// TIA Portal project "ENSACADPORA_030924" (V18)

(* hardware
DEVICE "SIMATIC 1200 station_1"  S7-1200 Station
   slot 0: "S7-1200 rack"  S7-1200 Rack  Rack  V1.0
   slot 1: "Master"  CPU 1212C DC/DC/Rly  6ES7 212-1HE40-0XB0  V4.5
   slot 2: "DI 8x24VDC/DQ 8xRelay_1"  SM 1223 DI8/DQ8 x relay  6ES7 223-1PH32-0XB0  V2.0
   slot 101: "CM 1241 (RS422/485)_1"  6ES7 241-1CH32-0XB0  V2.2
*)

// ===== PLC "Master"  CPU 1212C DC/DC/Rly =====

VAR_GLOBAL   // PLC tag table "Default tag table"
   "Input_IniciarLLenado" AT %I0.0 : Bool;
   "Input_PararLLenado" AT %I0.1 : Bool;
   "Input_ParoEmergencia" AT %I0.2 : Bool;
   "Input_SensorInicioPistonComp" AT %I0.3 : Bool;
   "Input_SensorFinPistonComp" AT %I0.4 : Bool;
   "COM_ACTIVA" AT %M113.0 : Bool;
   "StepCom" AT %MB57 : Byte;
   "System_Byte" AT %MB58 : Byte;
   "FirstScan" AT %M50.0 : Bool;
   "DiagStatusUpdate" AT %M50.1 : Bool;
   "AlwaysTRUE" AT %M50.2 : Bool;
   "AlwaysFALSE" AT %M50.3 : Bool;
   "FrmHmi_EncenderMotorHelicoidal" AT %M60.0 : Bool;
   "FrmHmi_ApagarMotorHelicoidal" AT %M60.1 : Bool;
   "FrmHmi_ResetFallas" AT %M61.0 : Bool;
   "Refe_Frec_FromHmi_ToVdf" AT %MW0 : Int;
   "AuxIn_IniciarLLenado" AT %M56.0 : Bool;
   "AuxIn_PararLLenado" AT %M56.1 : Bool;
   "AuxIn_ParoEmergancia" AT %M56.2 : Bool;
   "AuxIn_SensorInicioComp" AT %M56.3 : Bool;
   "AuxIn_SensorFinalComp" AT %M56.4 : Bool;
   "FrmHmi_ModManual" AT %M63.0 : Bool;
   "FrmHmi_Automatico" AT %M63.1 : Bool;
   "FrmHmi_ActivarPistonCompuerta" AT %M60.2 : Bool;
   "FrmHmi_DesactivarPistonCompuerta" AT %M60.3 : Bool;
   "Aux_Modo_Manual" AT %M64.0 : Bool;
   "Aux_Modo_Auto" AT %M64.1 : Bool;
   "SetPoitKilos" AT %MD4 : Real;
   "FrmHmi_HacerZeroBas" AT %M60.7 : Bool;
   "PB POLARIDAD" AT %M65.0 : Bool;
   "BAS ESTABLE" AT %M65.1 : Bool;
   "BAS UNDERLOAD" AT %M65.2 : Bool;
   "BAS OVERLOAD" AT %M65.3 : Bool;
   "BAS TARA HECHA" AT %M65.4 : Bool;
   "BAS EN ZERO" AT %M65.5 : Bool;
   "PESO NETO BASCULA" AT %MD44 : Real;
   "FrmHmi_ActivarModBarrido" AT %M63.2 : Bool;
   "OUT_VDF_MOTOR" AT %Q0.0 : Bool;
   "OUT_VIBRADOR" AT %Q0.2 : Bool;
   "OUT_COMPUERTA_ABIERTA" AT %Q0.1 : Bool;
   "FrmHmi_EncenderVibradorEnsacadora" AT %M60.4 : Bool;
   "FrmHmi_ApagarVibradorEnsacadora" AT %M60.5 : Bool;
   "Aux_Modo_Barrido" AT %M64.2 : Bool;
   "FrmHmi_DesactivarModBarrido" AT %M63.3 : Bool;
   "AUX_OUT_MOTOR" AT %M66.0 : Bool;
   "AUX_OUT_VIBRADOR" AT %M66.1 : Bool;
   "AUX_OUT_COMPUERTA_ABIERTA" AT %M66.2 : Bool;
   "AUX_OUT_MOTOR_BARRIDO" AT %M66.3 : Bool;
   "AUX_OUT_VIBRADOR_BARRIDO" AT %M66.4 : Bool;
   "AUX_OUT_COMPUERTA_BARRIDO_ABIERTA" AT %M66.5 : Bool;
   "ESTATUS_OPERACION" AT %MW8 : Int;
   "FrmHmi_Barrido" AT %M63.4 : Bool;
   "AUX_PARO_EMERGENCIA" AT %M61.1 : Bool;
   "INCIAR CICLO" AT %M62.0 : Bool;
   "APAGAR CICLO" AT %M62.1 : Bool;
   "Aux_Reset_Ciclo" AT %M64.3 : Bool;
   "Aux Error COM bascula" AT %M64.4 : Bool;
   "Aux iniciar ciclo" AT %M64.5 : Bool;
   "STEP BASCULA" AT %MW10 : Int;
   "Aux Valvula compuerta de carga_abierta" AT %M64.6 : Bool;
   "Abriendo compuerta de carga" AT %M67.0 : Bool;
   "Aux Sensor Compuerta Carga Abierta" AT %M64.7 : Bool;
   "pasa o no pasa" AT %MW12 : Int;
   "PESO NETO" AT %MD40 : Real;
   "TARAR" AT %MD36 : Real;
   "aux zero manual" AT %M60.6 : Bool;
   "AUX_HACER_ZERO" AT %M65.6 : Bool;
   "ZERO RES" AT %M65.7 : Bool;
   "SETPOINT" AT %MW2 : Int;
   "ACTIVAR MOTOR" AT %M66.6 : Bool;
   "PUNTO DE CORTE" AT %MD32 : Real;
   "% Corte VFD Grueso" AT %MW14 : Int;
   "Frec Max Mot Fino" AT %MW16 : Int;
   "OUT FRECU PARA VDF FINO" AT %MW18 : Int;
   "DIFERENCIA" AT %MD28 : Real;
   "DIV" AT %MD20 : Real;
   "FILTRO" AT %MD24 : Real;
   "Aux falla arranque VDF" AT %M56.5 : Bool;
   "Aux falla compuerta abierta al dosificar" AT %M56.6 : Bool;
   "ENCENDER VDF" AT %M62.2 : Bool;
   "APAGAR VDF" AT %M62.3 : Bool;
   "MAYOR QUE SETPOINT" AT %MD48 : Real;
   "MENOR QUE SETPOINT" AT %MD52 : Real;
   "DEFAULT CORTE SETPOINT" AT %MD68 : Real;
   "LISTO PARA PONER SACO" AT %M62.4 : Bool;
   "ESPERANDO QUE PONGAN EL COSTAL" AT %M62.5 : Bool;
   "Aux Sensor Sujetador Cerrado" AT %M59.0 : Bool;
   "GRAMOS DESDE HMI" AT %MW76 : Word;
   "GRAMOS SECUENCIA" AT %MD72 : Real;
   "Input_IniciarLLenado_v" AT %M80.0 : Bool;
   "Input_PararLLenado_v" AT %M80.1 : Bool;
   "Input_ParoEmergencia_v" AT %M80.2 : Bool;
   "Input_SensorInicioPistonComp_v" AT %M80.3 : Bool;
   "Input_SensorFinPistonComp_v" AT %M80.4 : Bool;
   "input_sensor_compuerta_descarga_v" AT %M80.5 : Bool;
   "input_sensor_sujetador_cerrado_v" AT %M80.6 : Bool;
   "input_valvula_compuerta_descarga_v" AT %M80.7 : Bool;
   "AUX_TIME_VIBRADOR" AT %M66.7 : Bool;
   "AUX_OUT_VIBRADOR_TIME" AT %M67.1 : Bool;
   "Falla al cerrar compuerta descarga" AT %M78.0 : Bool;
   "Falla al abrir compuerta descarga" AT %M78.1 : Bool;
   "Falla en el tiempo de vibrador" AT %M78.2 : Bool;
   "Fallas activas" AT %M78.3 : Bool;
   "RESETEAR FALLAS" AT %M61.2 : Bool;
   "TIEMPO ENCENDIDO VIBRADOR" AT %MD84 : DInt;
   "TIEMPO APAGADO VIBRADOR" AT %MD88 : DInt;
   "VerCalibracion" AT %M79.0 : Bool;
   "Reset_Indicador" AT %M79.1 : Bool;
   "CapturarZeroBascula" AT %M79.2 : Bool;
   "CapturarPesoEnBascula" AT %M79.3 : Bool;
   "GuardarCalibracion" AT %M79.4 : Bool;
   "CancelarCalibracion" AT %M79.5 : Bool;
   "ConfirmPesoParaCalibrar" AT %M79.6 : Bool;
   "EnviarPesoA_Calibrar" AT %M79.7 : Bool;
   "Timer_fallas_on" AT %M59.2 : Bool;
   "Timer_fallas_off" AT %M59.1 : Bool;
   "bits_contador_timer_on" AT %M114.0 : Bool;
   "bits_contador_timer_off" AT %M114.1 : Bool;
   "RESET_CONTADOR" AT %M114.2 : Bool;
   "CONTADOR" AT %MD116 : DInt;
   "PESO_PARA_CALIBRAR" AT %MD92 : DInt;
   "No se puede iniciar en cero" AT %M78.4 : Bool;
   "OUT_COMPUERTA_CERRADA" AT %Q0.3 : Bool;
   "ERROR EN EL MODBUS" AT %M112.0 : Bool;
   "AUXILIAR ERROR EN EL MODBUS" AT %M112.1 : Bool;
   "ERROR EN EL VARIADOR" AT %M112.2 : Bool;
   "AUXILIAR ERROR EN EL VARIADOR" AT %M112.3 : Bool;
   "direccion_byte_python" AT %MB115 : Byte;
   "Tag_1" AT %MD120 : DInt;
   "Tag_2" AT %MD124 : DInt;
END_VAR

TYPE "typeModbusCommLoad"
VERSION : 0.1
   STRUCT
      done : Bool := FALSE;   // Boolean indicating completion without error
      error : Bool := FALSE;   // Boolean indicating completion with error
      status : Word := W#16#0;   // Status or error code of the completed operation
      errorStatus : Word := W#16#0;   // Error code of the faulty operation
      doneStored : Bool := FALSE;   // Stored boolean indicating completion without error
   END_STRUCT;
END_TYPE

TYPE "typeModbusMaster"
VERSION : 0.1
   STRUCT
      req : Bool := FALSE;   // The enable to initiate a Modbus master request
      mbAddr : UInt;   // The station address of the Modbus slave
      mode : USInt := 0;   // Specifies a read, write, or diagnostic operation
      dataAddr : UDInt := 0;   // The Modbus data address
      dataLen : UInt := 0;   // The Modbus data length
      done : Bool := FALSE;   // Boolean indicating completion without error
      busy : Bool := FALSE;   // Boolean indicating operation in progress
      error : Bool := FALSE;   // Boolean indicating completion with error
      status : Word := W#16#0;   // Status or error code of the completed operation
      errorStatus : Word := W#16#0;   // Error code of the faulty operation
   END_STRUCT;
END_TYPE

TYPE "typeDataPtr"
VERSION : 0.1
   STRUCT
      data : Array[0..11] of Int;
   END_STRUCT;
END_TYPE

DATA_BLOCK "MasterData"   // DB1
{ S7_Optimized_Access := 'FALSE' }
VERSION : 0.1
   VAR
      "WRITE BASCULA" : Array[0..3] of Int;
      "READ BASCULA" : Array[0..10] of Int;
      "STATUS CAL" : Array[0..1] of Int;
      "WRITE VDF MOTOR" : Array[0..1] of Int;
      "READ VDF MOTOR" : Array[0..10] of Int;
      "PESO CALIBRAR" : Array[0..1] of Int;
      "LEER PESO CALIBRAR" : Array[0..1] of Int;
   END_VAR
BEGIN
END_DATA_BLOCK

DATA_BLOCK "Process"   // DB3
{ S7_Optimized_Access := 'TRUE' }
VERSION : 0.1
   VAR
      "step" : USInt := 1;
      edge : Bool := false;
      modbusMaster : "typeModbusMaster";
      modbusCommLoad : "typeModbusCommLoad";
   END_VAR
BEGIN
   modbusMaster.mbAddr := 2;
   modbusMaster.dataLen := 2;
END_DATA_BLOCK

DATA_BLOCK "HACER TARA_DB"   // DB6
{ S7_Optimized_Access := 'TRUE' }
VERSION : 0.1
// stored: InstanceOfName HACER TARA
"HACER TARA"
BEGIN
END_DATA_BLOCK

DATA_BLOCK "PORCENTAJE DE CORTE VDF GRUESO_DB_DB"   // DB9
{ S7_Optimized_Access := 'TRUE' }
VERSION : 0.1
// stored: InstanceOfName PORCENTAJE DE CORTE VDF GRUESO_DB
"PORCENTAJE DE CORTE VDF GRUESO_DB"
BEGIN
END_DATA_BLOCK

DATA_BLOCK "HACER TARA_DB_1"   // DB11
{ S7_Optimized_Access := 'TRUE' }
VERSION : 0.1
// stored: InstanceOfName HACER TARA
"HACER TARA"
BEGIN
END_DATA_BLOCK

DATA_BLOCK "python"   // DB23
{ S7_Optimized_Access := 'FALSE' }
VERSION : 0.1
   VAR
      estatus : Array[0..1] of Bool;
      "Contador y Estatus" : Array[0..1] of Int;
      Bascula : Array[0..0] of Real;
   END_VAR
BEGIN
   "Contador y Estatus"[0] := 0;
   estatus[0] := True;
   estatus[1] := False;
END_DATA_BLOCK

// folder: System blocks/Program resources

DATA_BLOCK "IEC_Timer_0_DB"   // DB2
{ S7_Optimized_Access := 'TRUE' }
AUTHOR : Simatic
FAMILY : IEC
NAME : IEC_TMR
VERSION : 1.0
// stored: InstanceOfName IEC_TIMER
"IEC_TIMER"
BEGIN
END_DATA_BLOCK

DATA_BLOCK "IEC_Timer_0_DB_1"   // DB7
{ S7_Optimized_Access := 'TRUE' }
AUTHOR : Simatic
FAMILY : IEC
NAME : IEC_TMR
VERSION : 1.0
// stored: InstanceOfName IEC_TIMER
"IEC_TIMER"
BEGIN
END_DATA_BLOCK

DATA_BLOCK "IEC_Timer_0_DB_2"   // DB8
{ S7_Optimized_Access := 'TRUE' }
AUTHOR : Simatic
FAMILY : IEC
NAME : IEC_TMR
VERSION : 1.0
// stored: InstanceOfName IEC_TIMER
"IEC_TIMER"
BEGIN
END_DATA_BLOCK

DATA_BLOCK "IEC_Timer_0_DB_3"   // DB10
{ S7_Optimized_Access := 'TRUE' }
AUTHOR : Simatic
FAMILY : IEC
NAME : IEC_TMR
VERSION : 1.0
// stored: InstanceOfName IEC_TIMER
"IEC_TIMER"
BEGIN
END_DATA_BLOCK

DATA_BLOCK "IEC_Timer_0_DB_4"   // DB12
{ S7_Optimized_Access := 'TRUE' }
AUTHOR : Simatic
FAMILY : IEC
NAME : IEC_TMR
VERSION : 1.0
// stored: InstanceOfName IEC_TIMER
"IEC_TIMER"
BEGIN
END_DATA_BLOCK

DATA_BLOCK "IEC_Timer_0_DB_5"   // DB13
{ S7_Optimized_Access := 'TRUE' }
AUTHOR : Simatic
FAMILY : IEC
NAME : IEC_TMR
VERSION : 1.0
// stored: InstanceOfName IEC_TIMER
"IEC_TIMER"
BEGIN
END_DATA_BLOCK

DATA_BLOCK "IEC_Timer_0_DB_6"   // DB14
{ S7_Optimized_Access := 'TRUE' }
AUTHOR : Simatic
FAMILY : IEC
NAME : IEC_TMR
VERSION : 1.0
// stored: InstanceOfName IEC_TIMER
"IEC_TIMER"
BEGIN
END_DATA_BLOCK

DATA_BLOCK "IEC_Timer_0_DB_7"   // DB15
{ S7_Optimized_Access := 'TRUE' }
AUTHOR : Simatic
FAMILY : IEC
NAME : IEC_TMR
VERSION : 1.0
// stored: InstanceOfName IEC_TIMER
"IEC_TIMER"
BEGIN
END_DATA_BLOCK

DATA_BLOCK "IEC_Timer_0_DB_8"   // DB16
{ S7_Optimized_Access := 'TRUE' }
AUTHOR : Simatic
FAMILY : IEC
NAME : IEC_TMR
VERSION : 1.0
// stored: InstanceOfName IEC_TIMER
"IEC_TIMER"
BEGIN
END_DATA_BLOCK

DATA_BLOCK "IEC_Timer_0_DB_9"   // DB17
{ S7_Optimized_Access := 'TRUE' }
AUTHOR : Simatic
FAMILY : IEC
NAME : IEC_TMR
VERSION : 1.0
// stored: InstanceOfName IEC_TIMER
"IEC_TIMER"
BEGIN
END_DATA_BLOCK

DATA_BLOCK "IEC_Timer_0_DB_10"   // DB18
{ S7_Optimized_Access := 'TRUE' }
AUTHOR : Simatic
FAMILY : IEC
NAME : IEC_TMR
VERSION : 1.0
// stored: InstanceOfName IEC_TIMER
"IEC_TIMER"
BEGIN
END_DATA_BLOCK

DATA_BLOCK "IEC_Counter_0_DB"   // DB19
{ S7_Optimized_Access := 'TRUE' }
AUTHOR : Simatic
FAMILY : IEC
NAME : CNTR
VERSION : 1.0
// stored: InstanceOfName IEC_COUNTER
"IEC_COUNTER"
BEGIN
END_DATA_BLOCK

DATA_BLOCK "IEC_Timer_0_DB_11"   // DB20
{ S7_Optimized_Access := 'TRUE' }
AUTHOR : Simatic
FAMILY : IEC
NAME : IEC_TMR
VERSION : 1.0
// stored: InstanceOfName IEC_TIMER
"IEC_TIMER"
BEGIN
END_DATA_BLOCK

DATA_BLOCK "IEC_Timer_0_DB_12"   // DB21
{ S7_Optimized_Access := 'TRUE' }
AUTHOR : Simatic
FAMILY : IEC
NAME : IEC_TMR
VERSION : 1.0
// stored: InstanceOfName IEC_TIMER
"IEC_TIMER"
BEGIN
END_DATA_BLOCK

DATA_BLOCK "IEC_Timer_0_DB_13"   // DB22
{ S7_Optimized_Access := 'TRUE' }
AUTHOR : Simatic
FAMILY : IEC
NAME : IEC_TMR
VERSION : 1.0
// stored: InstanceOfName IEC_TIMER
"IEC_TIMER"
BEGIN
END_DATA_BLOCK

// folder: (top level)

FUNCTION_BLOCK "HACER TARA"   // FB1, LAD
{ S7_Optimized_Access := 'TRUE' }
VERSION : 0.1
   VAR_INPUT
      TARAR2 : Bool;
      TARAR1 : Bool;
   END_VAR
   VAR_OUTPUT
      "PESO NETO TARA" : Real;
   END_VAR
   VAR_TEMP
      TARA : Real;
      TA : Bool;
      TA2 : Bool;
      available : Bool;
   END_VAR
   VAR_TEMP   // added for the SCL form of the ladder/FBD networks
      _w1 : Bool;
   END_VAR
BEGIN

REGION Network 1: HACER TARA
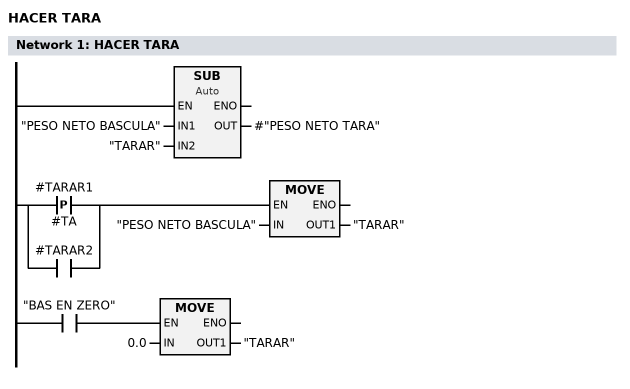
   RUNG wire#powerrail
      Sub(in1 := "PESO NETO BASCULA", in2 := "TARAR", out => #"PESO NETO TARA")
   END_RUNG
   RUNG wire#powerrail
      P_Contact(operand := #TARAR1, bit := #TA)
      wire#w1
      Move(in := "PESO NETO BASCULA", out1 => "TARAR")
   END_RUNG
   RUNG wire#powerrail
      Contact( #TARAR2 )
   END_RUNG wire#w1
   RUNG wire#powerrail
      Contact( "BAS EN ZERO" )
      Move(in := 0.0, out1 => "TARAR")
   END_RUNG
   // the same network as SCL:
   #"PESO NETO TARA" := "PESO NETO BASCULA" - "TARAR";
   #_w1 := #TARAR1 AND NOT #TA;   // rising edge of #TARAR1
   #TA := #TARAR1;
   IF #_w1 OR #TARAR2 THEN "TARAR" := "PESO NETO BASCULA"; END_IF;
   IF "BAS EN ZERO" THEN "TARAR" := 0.0; END_IF;
END_REGION
END_FUNCTION_BLOCK

FUNCTION_BLOCK "PORCENTAJE DE CORTE VDF GRUESO_DB"   // FB2, LAD
{ S7_Optimized_Access := 'TRUE' }
VERSION : 0.1
   VAR_INPUT
      "Set point" : Int;
      "% De Corte" : Int;
      PesoNeto : Real;
   END_VAR
   VAR_OUTPUT
      "Cantidad a cortar" : Real;
      "Bit OFF VDF Grueso" : Bool;
   END_VAR
   VAR_TEMP
      MULTI : Int;
   END_VAR
BEGIN

REGION Network 1: PORCENTAJE DE CORTE
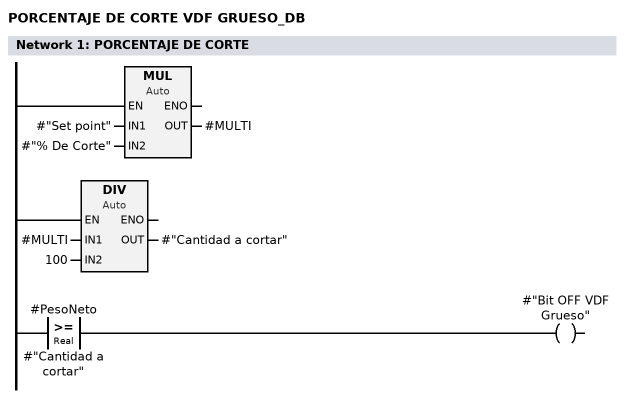
   RUNG wire#powerrail
      Mul(in1 := #"Set point", in2 := #"% De Corte", out => #MULTI)
   END_RUNG
   RUNG wire#powerrail
      Div(in1 := #MULTI, in2 := 100, out => #"Cantidad a cortar")
   END_RUNG
   RUNG wire#powerrail
      { S7_Templates := "SrcType := Real" } GE_Contact(in1 := #PesoNeto, in2 := #"Cantidad a cortar")
      Coil( #"Bit OFF VDF Grueso" )
   END_RUNG
   // the same network as SCL:
   #MULTI := #"Set point" * #"% De Corte";
   #"Cantidad a cortar" := #MULTI / 100;
   #"Bit OFF VDF Grueso" := #PesoNeto >= #"Cantidad a cortar";
END_REGION
END_FUNCTION_BLOCK

ORGANIZATION_BLOCK "1- COMUNICACION MODBUS"   // OB1, LAD, ProgramCycle
TITLE = PROGRAMACION CENTRIFUGAS
{ S7_Optimized_Access := 'TRUE' }
VERSION : 0.1
   VAR_INPUT
      Initial_Call : Bool;   // Initial call of this OB
      Remanence : Bool;   // =True, if remanent data are available
   END_VAR
   VAR_TEMP
      OutFrecMot : Int;
      OutRefFrecMot : Int;
      OutCorrienteMot : Real;
      "Bits Bascula" : DInt;
      "weig neto" : Real;
   END_VAR
   VAR_TEMP   // added for the SCL form of the ladder/FBD networks
      _w1 : Bool;
   END_VAR
BEGIN

REGION Network 1: INICIALIZAR COMUNICACION
   // "Modbus_Master_DB".MB_DB (not "Modbus_Master_DB")
   // 16#81AA (Invalid operating mode) -> Modbus_Comm_Load_DB.MODE = Half duplex (RS485) two-wire mode. (4)
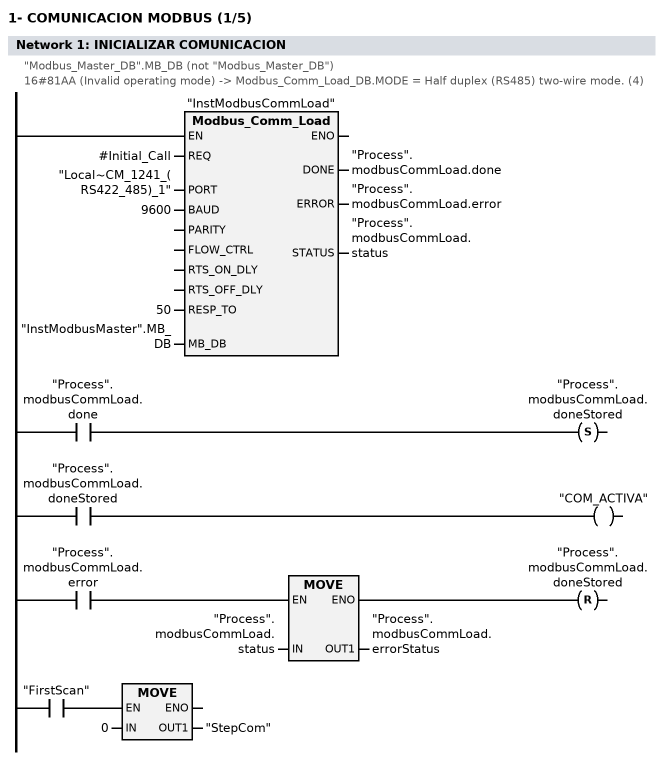
   // ENO of a box is taken as its EN; it also drops when the box reports an error
   "InstModbusCommLoad"(REQ := #Initial_Call,   // Modbus_Comm_Load
                        PORT := "Local~CM_1241_(RS422_485)_1",
                        BAUD := 9600,
                        RESP_TO := 50,
                        MB_DB := "InstModbusMaster".MB_DB,
                        DONE => "Process".modbusCommLoad.done,
                        ERROR => "Process".modbusCommLoad.error,
                        STATUS => "Process".modbusCommLoad.status);
   IF "Process".modbusCommLoad.done THEN "Process".modbusCommLoad.doneStored := TRUE; END_IF;
   "COM_ACTIVA" := "Process".modbusCommLoad.doneStored;
   IF "Process".modbusCommLoad.error THEN
       "Process".modbusCommLoad.errorStatus := "Process".modbusCommLoad.status;
       "Process".modbusCommLoad.doneStored := FALSE;
   END_IF;
   IF "FirstScan" THEN "StepCom" := 0; END_IF;
END_REGION

REGION Network 2: LEER--ESCRIBIR, BASCULA
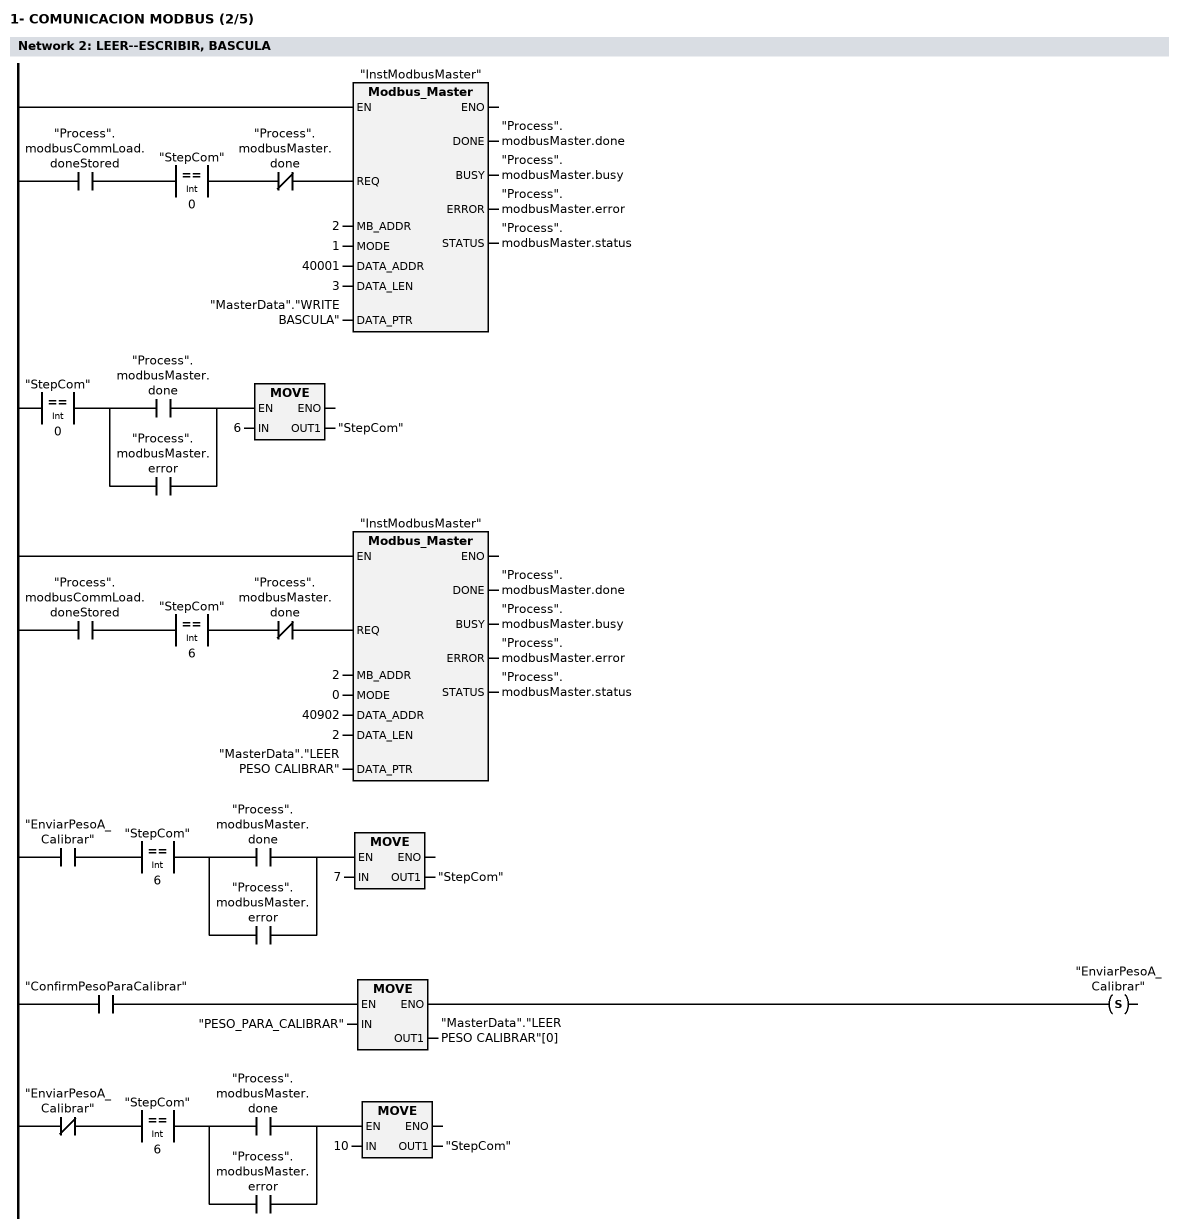
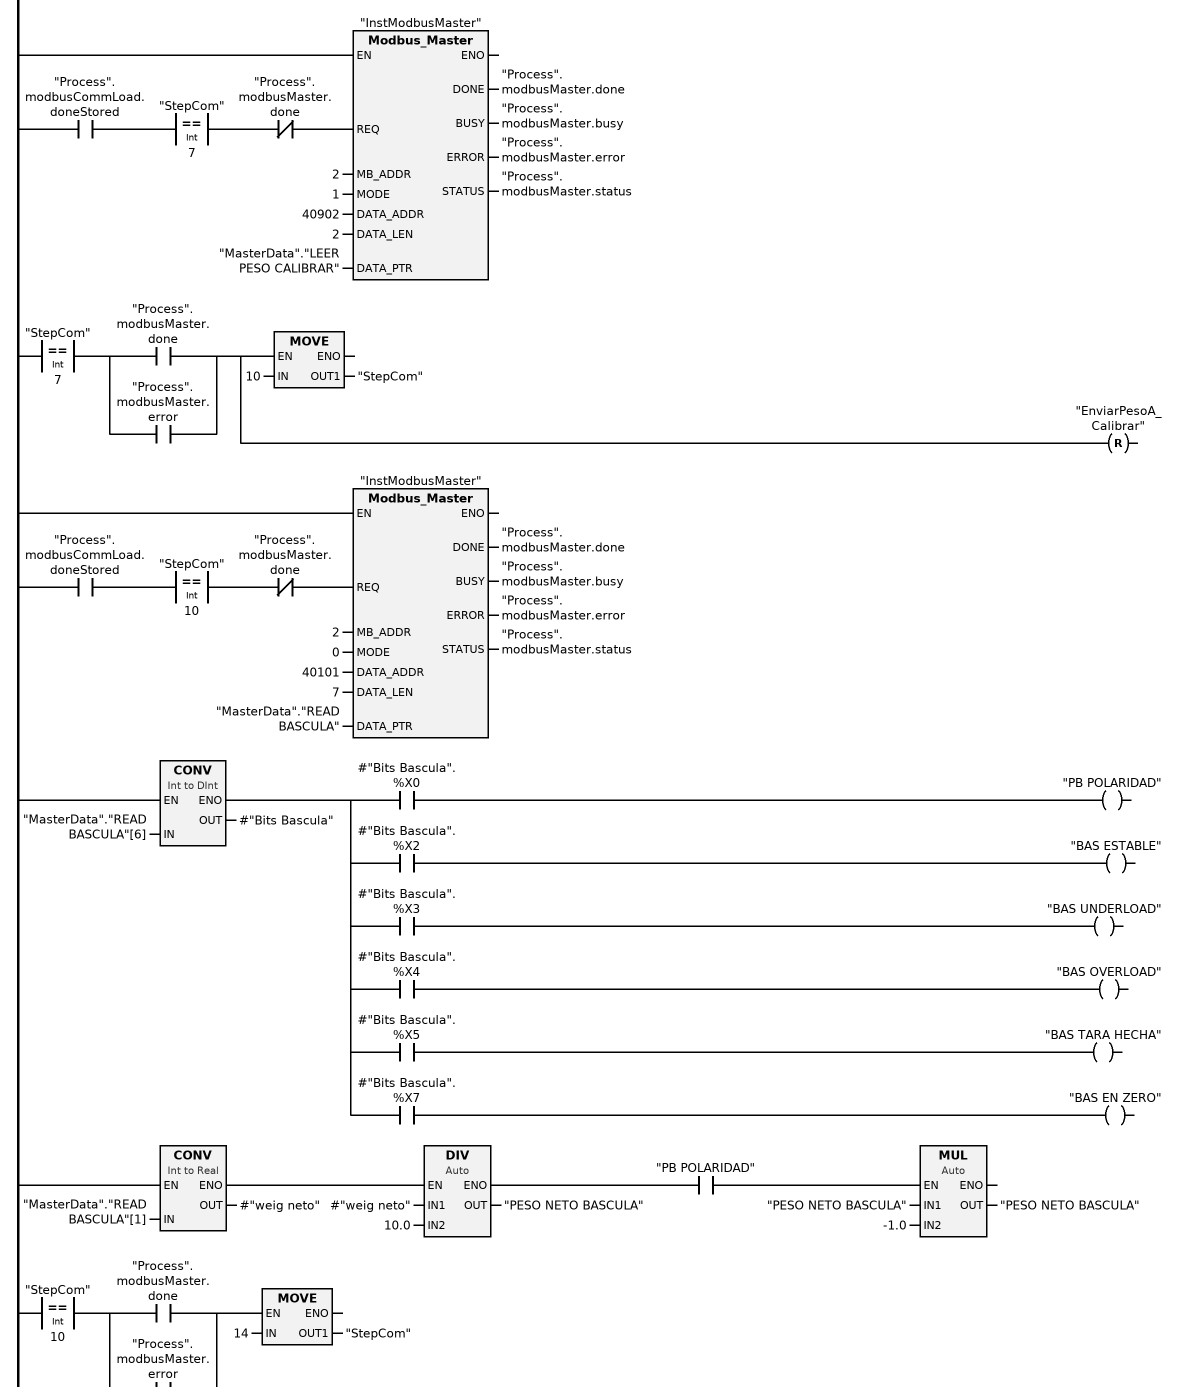
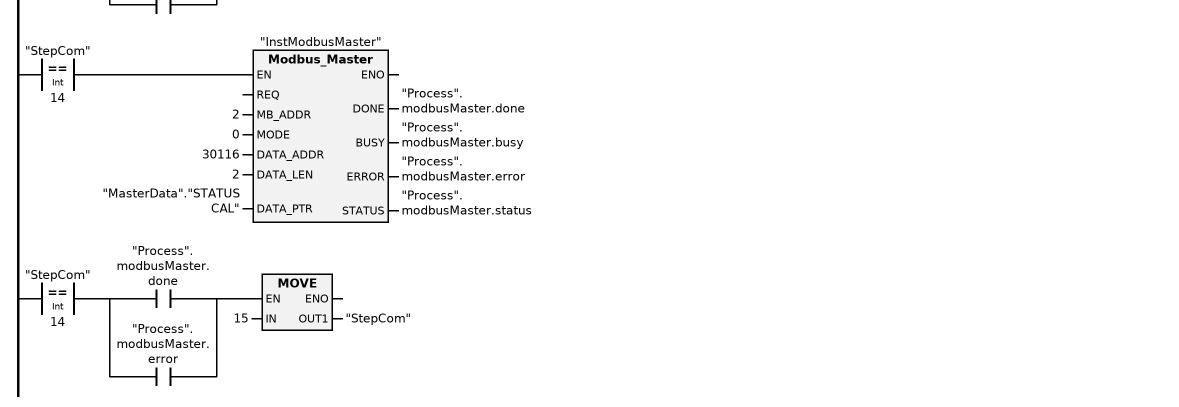
   "InstModbusMaster"(REQ := "Process".modbusCommLoad.doneStored AND ("StepCom" = 0) AND NOT "Process".modbusMaster.done,   // Modbus_Master
                      MB_ADDR := 2,
                      MODE := 1,
                      DATA_ADDR := 40001,
                      DATA_LEN := 3,
                      DATA_PTR := "MasterData"."WRITE BASCULA",
                      DONE => "Process".modbusMaster.done,
                      BUSY => "Process".modbusMaster.busy,
                      ERROR => "Process".modbusMaster.error,
                      STATUS => "Process".modbusMaster.status);
   IF ("StepCom" = 0) AND ("Process".modbusMaster.done OR "Process".modbusMaster.error) THEN
       "StepCom" := 6;
   END_IF;
   "InstModbusMaster"(REQ := "Process".modbusCommLoad.doneStored AND ("StepCom" = 6) AND NOT "Process".modbusMaster.done,   // Modbus_Master
                      MB_ADDR := 2,
                      MODE := 0,
                      DATA_ADDR := 40902,
                      DATA_LEN := 2,
                      DATA_PTR := "MasterData"."LEER PESO CALIBRAR",
                      DONE => "Process".modbusMaster.done,
                      BUSY => "Process".modbusMaster.busy,
                      ERROR => "Process".modbusMaster.error,
                      STATUS => "Process".modbusMaster.status);
   IF "EnviarPesoA_Calibrar" AND ("StepCom" = 6) AND ("Process".modbusMaster.done OR "Process".modbusMaster.error) THEN
       "StepCom" := 7;
   END_IF;
   IF "ConfirmPesoParaCalibrar" THEN
       "MasterData"."LEER PESO CALIBRAR"[0] := "PESO_PARA_CALIBRAR";
       "EnviarPesoA_Calibrar" := TRUE;
   END_IF;
   IF NOT "EnviarPesoA_Calibrar" AND ("StepCom" = 6) AND ("Process".modbusMaster.done OR "Process".modbusMaster.error) THEN
       "StepCom" := 10;
   END_IF;
   "InstModbusMaster"(REQ := "Process".modbusCommLoad.doneStored AND ("StepCom" = 7) AND NOT "Process".modbusMaster.done,   // Modbus_Master
                      MB_ADDR := 2,
                      MODE := 1,
                      DATA_ADDR := 40902,
                      DATA_LEN := 2,
                      DATA_PTR := "MasterData"."LEER PESO CALIBRAR",
                      DONE => "Process".modbusMaster.done,
                      BUSY => "Process".modbusMaster.busy,
                      ERROR => "Process".modbusMaster.error,
                      STATUS => "Process".modbusMaster.status);
   #_w1 := ("StepCom" = 7) AND ("Process".modbusMaster.done OR "Process".modbusMaster.error);
   IF #_w1 THEN
       "StepCom" := 10;
       "EnviarPesoA_Calibrar" := FALSE;
   END_IF;
   "InstModbusMaster"(REQ := "Process".modbusCommLoad.doneStored AND ("StepCom" = 10) AND NOT "Process".modbusMaster.done,   // Modbus_Master
                      MB_ADDR := 2,
                      MODE := 0,
                      DATA_ADDR := 40101,
                      DATA_LEN := 7,
                      DATA_PTR := "MasterData"."READ BASCULA",
                      DONE => "Process".modbusMaster.done,
                      BUSY => "Process".modbusMaster.busy,
                      ERROR => "Process".modbusMaster.error,
                      STATUS => "Process".modbusMaster.status);
   #"Bits Bascula" := INT_TO_DINT("MasterData"."READ BASCULA"[6]);
   "PB POLARIDAD" := #"Bits Bascula".%X0;
   "BAS ESTABLE" := #"Bits Bascula".%X2;
   "BAS UNDERLOAD" := #"Bits Bascula".%X3;
   "BAS OVERLOAD" := #"Bits Bascula".%X4;
   "BAS TARA HECHA" := #"Bits Bascula".%X5;
   "BAS EN ZERO" := #"Bits Bascula".%X7;
   #"weig neto" := INT_TO_REAL("MasterData"."READ BASCULA"[1]);
   "PESO NETO BASCULA" := #"weig neto" / 10.0;
   IF "PB POLARIDAD" THEN "PESO NETO BASCULA" := "PESO NETO BASCULA" * (-1.0); END_IF;
   IF ("StepCom" = 10) AND ("Process".modbusMaster.done OR "Process".modbusMaster.error) THEN
       "StepCom" := 14;
   END_IF;
   IF "StepCom" = 14 THEN
       "InstModbusMaster"(MB_ADDR := 2,   // Modbus_Master
                          MODE := 0,
                          DATA_ADDR := 30116,
                          DATA_LEN := 2,
                          DATA_PTR := "MasterData"."STATUS CAL",
                          DONE => "Process".modbusMaster.done,
                          BUSY => "Process".modbusMaster.busy,
                          ERROR => "Process".modbusMaster.error,
                          STATUS => "Process".modbusMaster.status);
   END_IF;
   IF ("StepCom" = 14) AND ("Process".modbusMaster.done OR "Process".modbusMaster.error) THEN
       "StepCom" := 15;
   END_IF;
END_REGION

REGION Network 3: FALLA EN LA BASCULA
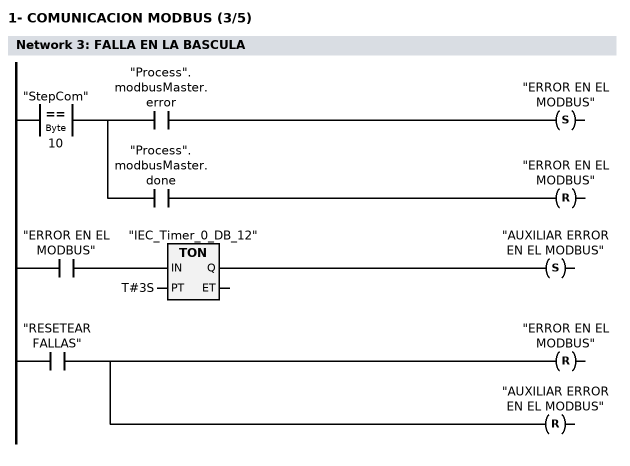
   #_w1 := "StepCom" = 10;
   IF #_w1 AND "Process".modbusMaster.error THEN "ERROR EN EL MODBUS" := TRUE; END_IF;
   IF #_w1 AND "Process".modbusMaster.done THEN "ERROR EN EL MODBUS" := FALSE; END_IF;
   "IEC_Timer_0_DB_12".TON(IN := "ERROR EN EL MODBUS", PT := T#3S);
   IF "IEC_Timer_0_DB_12".Q THEN "AUXILIAR ERROR EN EL MODBUS" := TRUE; END_IF;
   IF "RESETEAR FALLAS" THEN
       "ERROR EN EL MODBUS" := FALSE;
       "AUXILIAR ERROR EN EL MODBUS" := FALSE;
   END_IF;
END_REGION

REGION Network 4: LEER--ESCRIBIR, VDF MOTOR
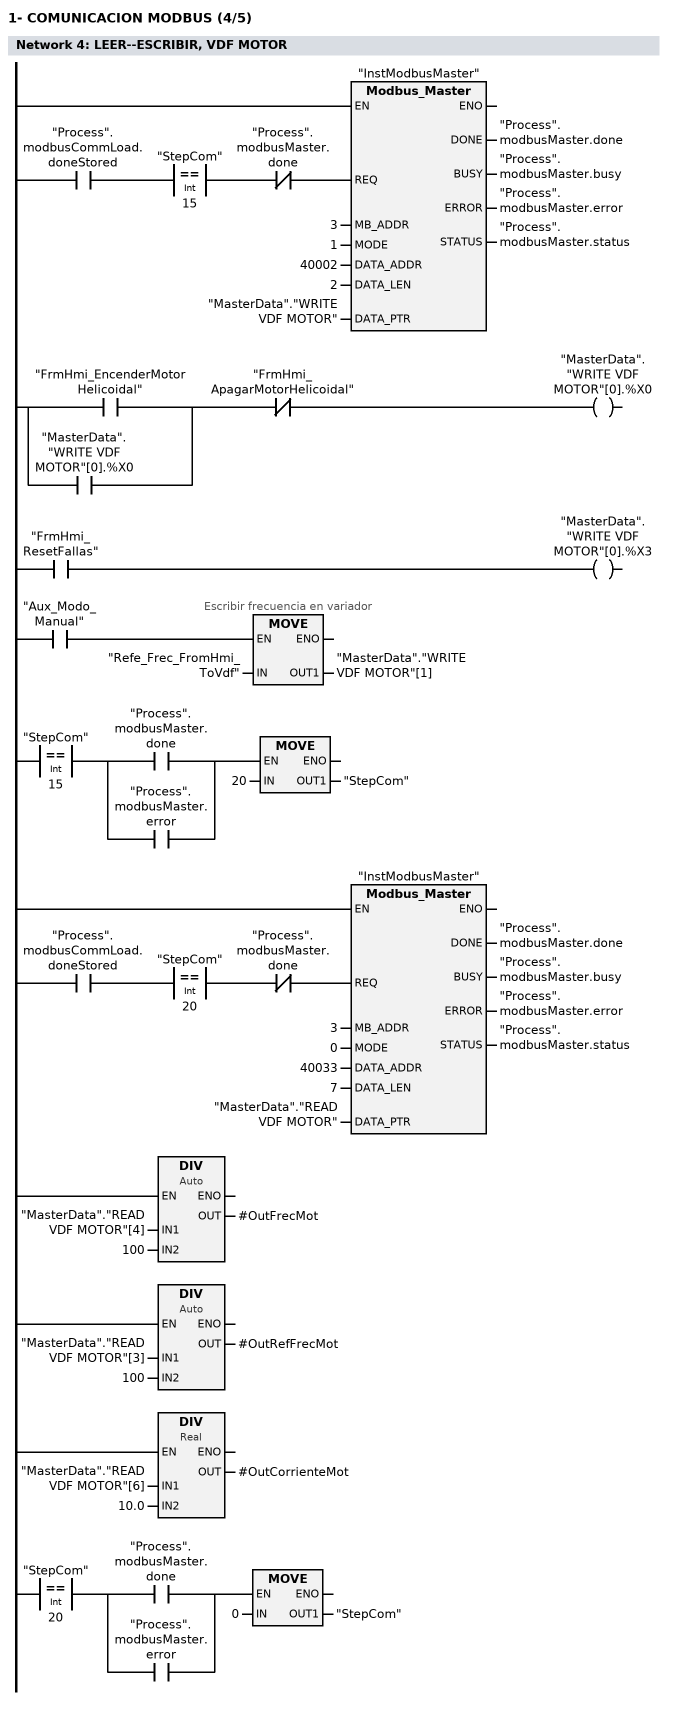
   "InstModbusMaster"(REQ := "Process".modbusCommLoad.doneStored AND ("StepCom" = 15) AND NOT "Process".modbusMaster.done,   // Modbus_Master
                      MB_ADDR := 3,
                      MODE := 1,
                      DATA_ADDR := 40002,
                      DATA_LEN := 2,
                      DATA_PTR := "MasterData"."WRITE VDF MOTOR",
                      DONE => "Process".modbusMaster.done,
                      BUSY => "Process".modbusMaster.busy,
                      ERROR => "Process".modbusMaster.error,
                      STATUS => "Process".modbusMaster.status);
   "MasterData"."WRITE VDF MOTOR"[0].%X0 := ("FrmHmi_EncenderMotorHelicoidal" OR "MasterData"."WRITE VDF MOTOR"[0].%X0) AND NOT "FrmHmi_ApagarMotorHelicoidal";
   "MasterData"."WRITE VDF MOTOR"[0].%X3 := "FrmHmi_ResetFallas";
   IF "Aux_Modo_Manual" THEN
       "MasterData"."WRITE VDF MOTOR"[1] := "Refe_Frec_FromHmi_ToVdf";   // Escribir frecuencia en variador
   END_IF;
   IF ("StepCom" = 15) AND ("Process".modbusMaster.done OR "Process".modbusMaster.error) THEN
       "StepCom" := 20;
   END_IF;
   "InstModbusMaster"(REQ := "Process".modbusCommLoad.doneStored AND ("StepCom" = 20) AND NOT "Process".modbusMaster.done,   // Modbus_Master
                      MB_ADDR := 3,
                      MODE := 0,
                      DATA_ADDR := 40033,
                      DATA_LEN := 7,
                      DATA_PTR := "MasterData"."READ VDF MOTOR",
                      DONE => "Process".modbusMaster.done,
                      BUSY => "Process".modbusMaster.busy,
                      ERROR => "Process".modbusMaster.error,
                      STATUS => "Process".modbusMaster.status);
   #OutFrecMot := "MasterData"."READ VDF MOTOR"[4] / 100;
   #OutRefFrecMot := "MasterData"."READ VDF MOTOR"[3] / 100;
   #OutCorrienteMot := "MasterData"."READ VDF MOTOR"[6] / 10.0;
   IF ("StepCom" = 20) AND ("Process".modbusMaster.done OR "Process".modbusMaster.error) THEN
       "StepCom" := 0;
   END_IF;
END_REGION

REGION Network 5: FALLA EN EL VARIADOR
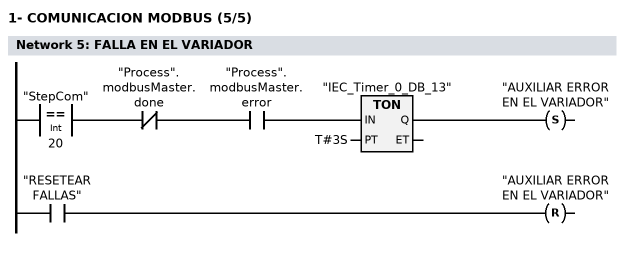
   "IEC_Timer_0_DB_13".TON(IN := ("StepCom" = 20) AND NOT "Process".modbusMaster.done AND "Process".modbusMaster.error,
                           PT := T#3S);
   IF "IEC_Timer_0_DB_13".Q THEN "AUXILIAR ERROR EN EL VARIADOR" := TRUE; END_IF;
   IF "RESETEAR FALLAS" THEN "AUXILIAR ERROR EN EL VARIADOR" := FALSE; END_IF;
END_REGION
END_ORGANIZATION_BLOCK

ORGANIZATION_BLOCK "2- ENTRADAS"   // OB123, LAD, ProgramCycle
TITLE = "Main Program Sweep (Cycle)"
{ S7_Optimized_Access := 'TRUE' }
VERSION : 0.1
   VAR_INPUT
      Initial_Call : Bool;   // Initial call of this OB
      Remanence : Bool;   // =True, if remanent data are available
   END_VAR
BEGIN

REGION Network 1: ENTRADAS FÍSICAS
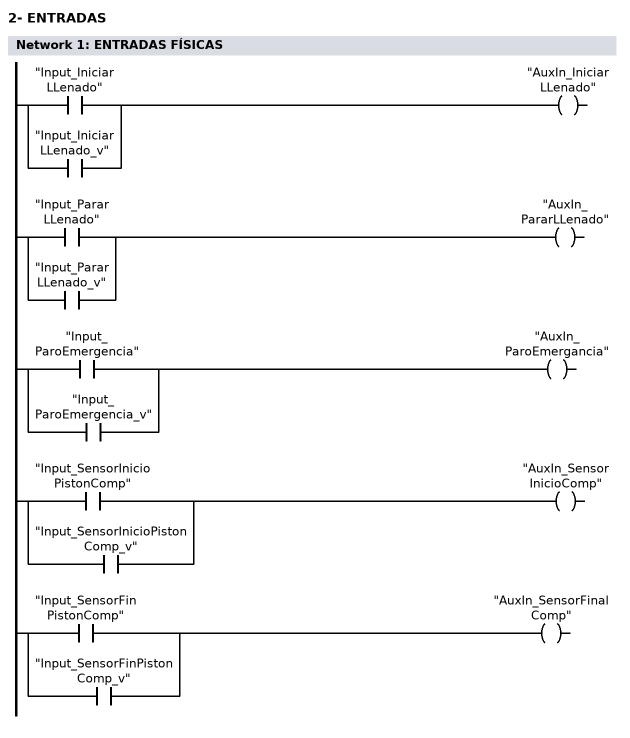
   RUNG wire#powerrail
      Contact( "Input_IniciarLLenado" )
      wire#w1
      Coil( "AuxIn_IniciarLLenado" )
   END_RUNG
   RUNG wire#powerrail
      Contact( "Input_IniciarLLenado_v" )
   END_RUNG wire#w1
   RUNG wire#powerrail
      Contact( "Input_PararLLenado" )
      wire#w2
      Coil( "AuxIn_PararLLenado" )
   END_RUNG
   RUNG wire#powerrail
      Contact( "Input_PararLLenado_v" )
   END_RUNG wire#w2
   RUNG wire#powerrail
      Contact( "Input_ParoEmergencia" )
      wire#w3
      Coil( "AuxIn_ParoEmergancia" )
   END_RUNG
   RUNG wire#powerrail
      Contact( "Input_ParoEmergencia_v" )
   END_RUNG wire#w3
   RUNG wire#powerrail
      Contact( "Input_SensorInicioPistonComp" )
      wire#w4
      Coil( "AuxIn_SensorInicioComp" )
   END_RUNG
   RUNG wire#powerrail
      Contact( "Input_SensorInicioPistonComp_v" )
   END_RUNG wire#w4
   RUNG wire#powerrail
      Contact( "Input_SensorFinPistonComp" )
      wire#w5
      Coil( "AuxIn_SensorFinalComp" )
   END_RUNG
   RUNG wire#powerrail
      Contact( "Input_SensorFinPistonComp_v" )
   END_RUNG wire#w5
   // the same network as SCL:
   "AuxIn_IniciarLLenado" := "Input_IniciarLLenado" OR "Input_IniciarLLenado_v";
   "AuxIn_PararLLenado" := "Input_PararLLenado" OR "Input_PararLLenado_v";
   "AuxIn_ParoEmergancia" := "Input_ParoEmergencia" OR "Input_ParoEmergencia_v";
   "AuxIn_SensorInicioComp" := "Input_SensorInicioPistonComp" OR "Input_SensorInicioPistonComp_v";
   "AuxIn_SensorFinalComp" := "Input_SensorFinPistonComp" OR "Input_SensorFinPistonComp_v";
END_REGION
END_ORGANIZATION_BLOCK

ORGANIZATION_BLOCK "3- LOGICA LLENADO"   // OB124, LAD, ProgramCycle
TITLE = "Main Program Sweep (Cycle)"
{ S7_Optimized_Access := 'TRUE' }
VERSION : 0.1
   VAR_INPUT
      Initial_Call : Bool;   // Initial call of this OB
      Remanence : Bool;   // =True, if remanent data are available
   END_VAR
   VAR_TEMP
      inhabilitar : Bool;
      AVAILABLE : Bool;
      frecoMOT : Int;
      "TIME ENCENDIDO" : Time;
      "TIME APAGADO" : Time;
      "RESULTADO ENCENDIDO" : Int;
      "RESULTADO APAGADO" : Int;
      status_operacion : Bool;
   END_VAR
   VAR_TEMP   // added for the SCL form of the ladder/FBD networks
      _w1 : Bool;
   END_VAR
BEGIN

REGION Network 1: MODO MANUAL, AUTOMATICO, BARRIDO
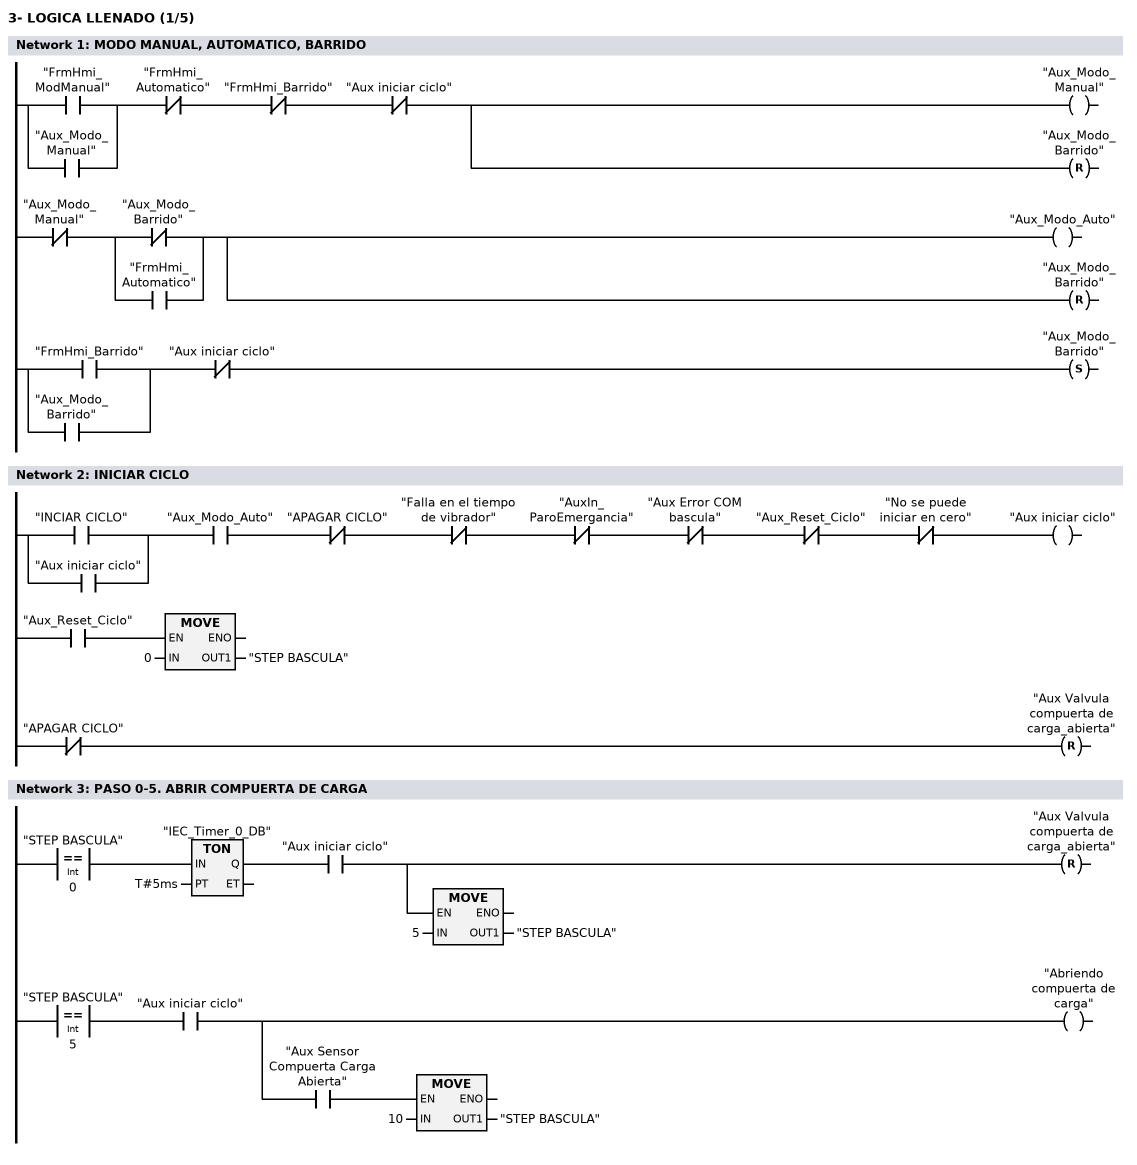
   RUNG wire#powerrail
      Contact( "FrmHmi_ModManual" )
      wire#w1
      I_Contact( "FrmHmi_Automatico" )
      I_Contact( "FrmHmi_Barrido" )
      I_Contact( "Aux iniciar ciclo" )
      wire#w2
      Coil( "Aux_Modo_Manual" )
   END_RUNG
   RUNG wire#powerrail
      Contact( "Aux_Modo_Manual" )
   END_RUNG wire#w1
   RUNG wire#w2
      R_Coil( "Aux_Modo_Barrido" )
   END_RUNG
   RUNG wire#powerrail
      I_Contact( "Aux_Modo_Manual" )
      wire#w3
      I_Contact( "Aux_Modo_Barrido" )
      wire#w4
      Coil( "Aux_Modo_Auto" )
   END_RUNG
   RUNG wire#w3
      Contact( "FrmHmi_Automatico" )
   END_RUNG wire#w4
   RUNG wire#w4
      R_Coil( "Aux_Modo_Barrido" )
   END_RUNG
   RUNG wire#powerrail
      Contact( "FrmHmi_Barrido" )
      wire#w5
      I_Contact( "Aux iniciar ciclo" )
      S_Coil( "Aux_Modo_Barrido" )
   END_RUNG
   RUNG wire#powerrail
      Contact( "Aux_Modo_Barrido" )
   END_RUNG wire#w5
   // the same network as SCL:
   "Aux_Modo_Manual" := ("FrmHmi_ModManual" OR "Aux_Modo_Manual") AND NOT "FrmHmi_Automatico" AND NOT "FrmHmi_Barrido" AND NOT "Aux iniciar ciclo";
   IF "Aux_Modo_Manual" THEN "Aux_Modo_Barrido" := FALSE; END_IF;
   "Aux_Modo_Auto" := NOT "Aux_Modo_Manual" AND (NOT "Aux_Modo_Barrido" OR "FrmHmi_Automatico");
   IF "Aux_Modo_Auto" THEN "Aux_Modo_Barrido" := FALSE; END_IF;
   IF ("FrmHmi_Barrido" OR "Aux_Modo_Barrido") AND NOT "Aux iniciar ciclo" THEN
       "Aux_Modo_Barrido" := TRUE;
   END_IF;
END_REGION

REGION Network 2: INICIAR CICLO
   RUNG wire#powerrail
      Contact( "INCIAR CICLO" )
      wire#w1
      Contact( "Aux_Modo_Auto" )
      I_Contact( "APAGAR CICLO" )
      I_Contact( "Falla en el tiempo de vibrador" )
      I_Contact( "AuxIn_ParoEmergancia" )
      I_Contact( "Aux Error COM bascula" )
      I_Contact( "Aux_Reset_Ciclo" )
      I_Contact( "No se puede iniciar en cero" )
      Coil( "Aux iniciar ciclo" )
   END_RUNG
   RUNG wire#powerrail
      Contact( "Aux iniciar ciclo" )
   END_RUNG wire#w1
   RUNG wire#powerrail
      Contact( "Aux_Reset_Ciclo" )
      Move(in := 0, out1 => "STEP BASCULA")
   END_RUNG
   RUNG wire#powerrail
      I_Contact( "APAGAR CICLO" )
      R_Coil( "Aux Valvula compuerta de carga_abierta" )
   END_RUNG
   // the same network as SCL:
   "Aux iniciar ciclo" := ("INCIAR CICLO" OR "Aux iniciar ciclo") AND "Aux_Modo_Auto" AND NOT "APAGAR CICLO" AND NOT "Falla en el tiempo de vibrador" AND NOT "AuxIn_ParoEmergancia" AND NOT "Aux Error COM bascula" AND NOT "Aux_Reset_Ciclo" AND NOT "No se puede iniciar en cero";
   IF "Aux_Reset_Ciclo" THEN "STEP BASCULA" := 0; END_IF;
   IF NOT "APAGAR CICLO" THEN "Aux Valvula compuerta de carga_abierta" := FALSE; END_IF;
END_REGION

REGION Network 3: PASO 0-5. ABRIR COMPUERTA DE CARGA
   "IEC_Timer_0_DB".TON(IN := "STEP BASCULA" = 0, PT := T#5ms);
   IF "IEC_Timer_0_DB".Q AND "Aux iniciar ciclo" THEN
       "Aux Valvula compuerta de carga_abierta" := FALSE;
       "STEP BASCULA" := 5;
   END_IF;
   "Abriendo compuerta de carga" := ("STEP BASCULA" = 5) AND "Aux iniciar ciclo";
   IF "Abriendo compuerta de carga" AND "Aux Sensor Compuerta Carga Abierta" THEN
       "STEP BASCULA" := 10;
   END_IF;
END_REGION

REGION Network 4: PASO 10. HACER TARA
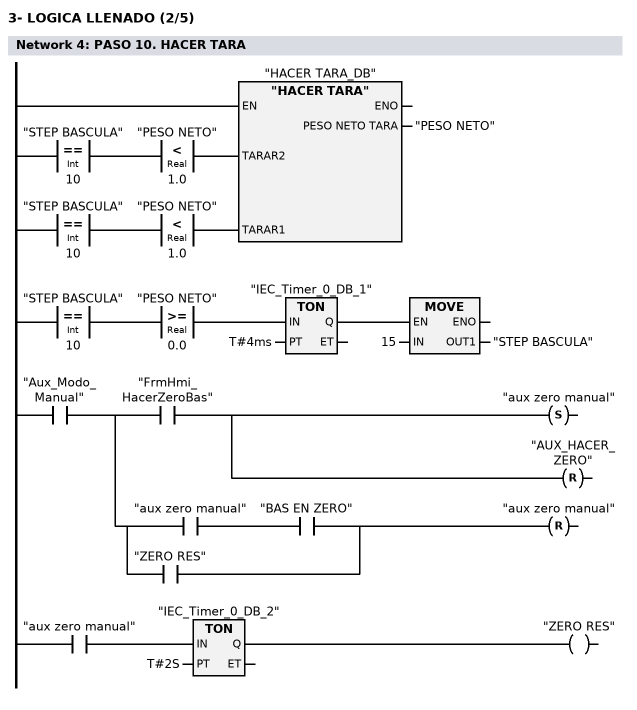
   "HACER TARA_DB"(TARAR2 := ("STEP BASCULA" = 10) AND ("PESO NETO" < 1.0),   // "HACER TARA"
                   TARAR1 := ("STEP BASCULA" = 10) AND ("PESO NETO" < 1.0),
                   "PESO NETO TARA" => "PESO NETO");
   "IEC_Timer_0_DB_1".TON(IN := ("STEP BASCULA" = 10) AND ("PESO NETO" >= 0.0), PT := T#4ms);
   IF "IEC_Timer_0_DB_1".Q THEN "STEP BASCULA" := 15; END_IF;
   IF "Aux_Modo_Manual" AND "FrmHmi_HacerZeroBas" THEN
       "aux zero manual" := TRUE;
       "AUX_HACER_ZERO" := FALSE;
   END_IF;
   IF "Aux_Modo_Manual" AND (("aux zero manual" AND "BAS EN ZERO") OR "ZERO RES") THEN
       "aux zero manual" := FALSE;
   END_IF;
   "IEC_Timer_0_DB_2".TON(IN := "aux zero manual", PT := T#2S);
   "ZERO RES" := "IEC_Timer_0_DB_2".Q;
END_REGION

REGION Network 5: PASO 15. ENCENDER Y APAGAR MOTORES
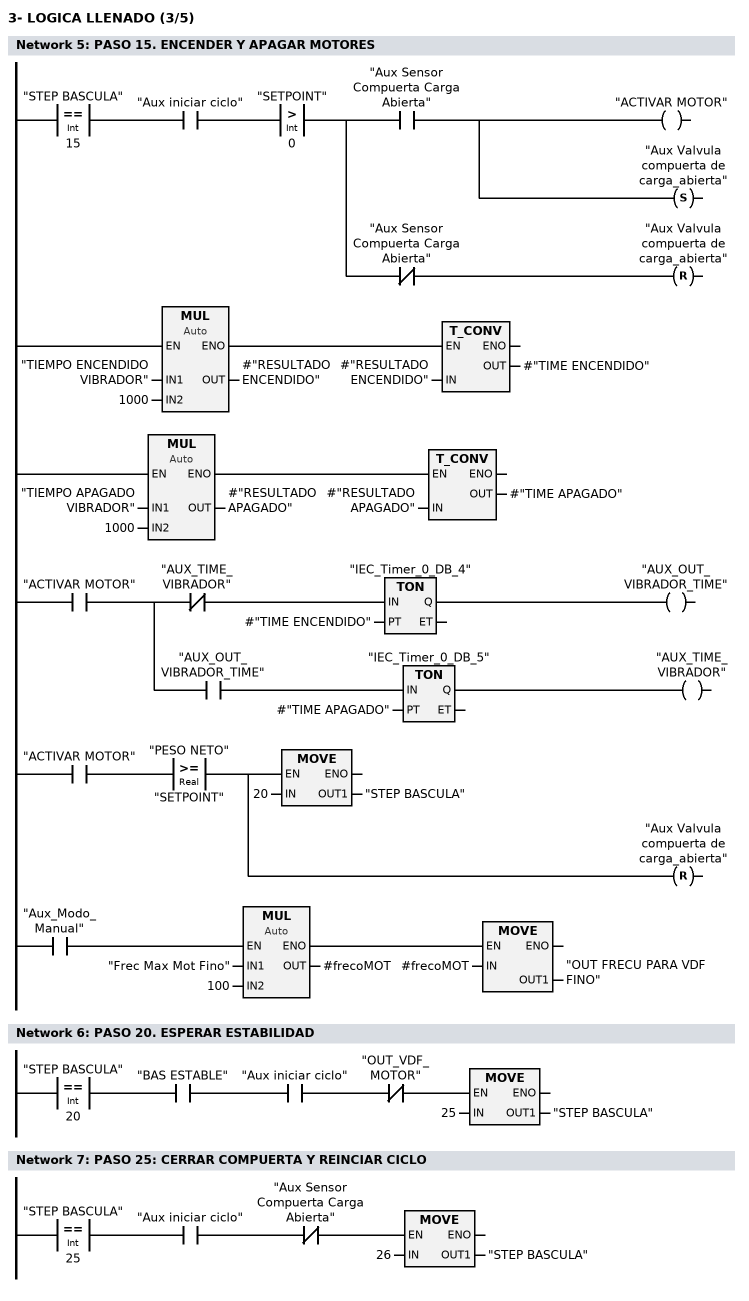
   #_w1 := ("STEP BASCULA" = 15) AND "Aux iniciar ciclo" AND ("SETPOINT" > 0);
   "ACTIVAR MOTOR" := #_w1 AND "Aux Sensor Compuerta Carga Abierta";
   IF "ACTIVAR MOTOR" THEN "Aux Valvula compuerta de carga_abierta" := TRUE; END_IF;
   IF #_w1 AND NOT "Aux Sensor Compuerta Carga Abierta" THEN
       "Aux Valvula compuerta de carga_abierta" := FALSE;
   END_IF;
   #"RESULTADO ENCENDIDO" := "TIEMPO ENCENDIDO VIBRADOR" * 1000;
   #"TIME ENCENDIDO" := T_CONV(IN := #"RESULTADO ENCENDIDO");
   #"RESULTADO APAGADO" := "TIEMPO APAGADO VIBRADOR" * 1000;
   #"TIME APAGADO" := T_CONV(IN := #"RESULTADO APAGADO");
   "IEC_Timer_0_DB_4".TON(IN := "ACTIVAR MOTOR" AND NOT "AUX_TIME_VIBRADOR", PT := #"TIME ENCENDIDO");
   "AUX_OUT_VIBRADOR_TIME" := "IEC_Timer_0_DB_4".Q;
   "IEC_Timer_0_DB_5".TON(IN := "ACTIVAR MOTOR" AND "AUX_OUT_VIBRADOR_TIME", PT := #"TIME APAGADO");
   "AUX_TIME_VIBRADOR" := "IEC_Timer_0_DB_5".Q;
   IF "ACTIVAR MOTOR" AND ("PESO NETO" >= "SETPOINT") THEN
       "STEP BASCULA" := 20;
       "Aux Valvula compuerta de carga_abierta" := FALSE;
   END_IF;
   IF "Aux_Modo_Manual" THEN
       #frecoMOT := "Frec Max Mot Fino" * 100;
       "OUT FRECU PARA VDF FINO" := #frecoMOT;
   END_IF;
END_REGION

REGION Network 6: PASO 20. ESPERAR ESTABILIDAD
   RUNG wire#powerrail
      { S7_Templates := "SrcType := Int" } EQ_Contact(in1 := "STEP BASCULA", in2 := 20)
      Contact( "BAS ESTABLE" )
      Contact( "Aux iniciar ciclo" )
      I_Contact( "OUT_VDF_MOTOR" )
      Move(in := 25, out1 => "STEP BASCULA")
   END_RUNG
   // the same network as SCL:
   IF ("STEP BASCULA" = 20) AND "BAS ESTABLE" AND "Aux iniciar ciclo" AND NOT "OUT_VDF_MOTOR" THEN
       "STEP BASCULA" := 25;
   END_IF;
END_REGION

REGION Network 7: PASO 25: CERRAR COMPUERTA Y REINCIAR CICLO
   RUNG wire#powerrail
      { S7_Templates := "SrcType := Int" } EQ_Contact(in1 := "STEP BASCULA", in2 := 25)
      Contact( "Aux iniciar ciclo" )
      I_Contact( "Aux Sensor Compuerta Carga Abierta" )
      Move(in := 26, out1 => "STEP BASCULA")
   END_RUNG
   // the same network as SCL:
   IF ("STEP BASCULA" = 25) AND "Aux iniciar ciclo" AND NOT "Aux Sensor Compuerta Carga Abierta" THEN
       "STEP BASCULA" := 26;
   END_IF;
END_REGION

REGION Network 8
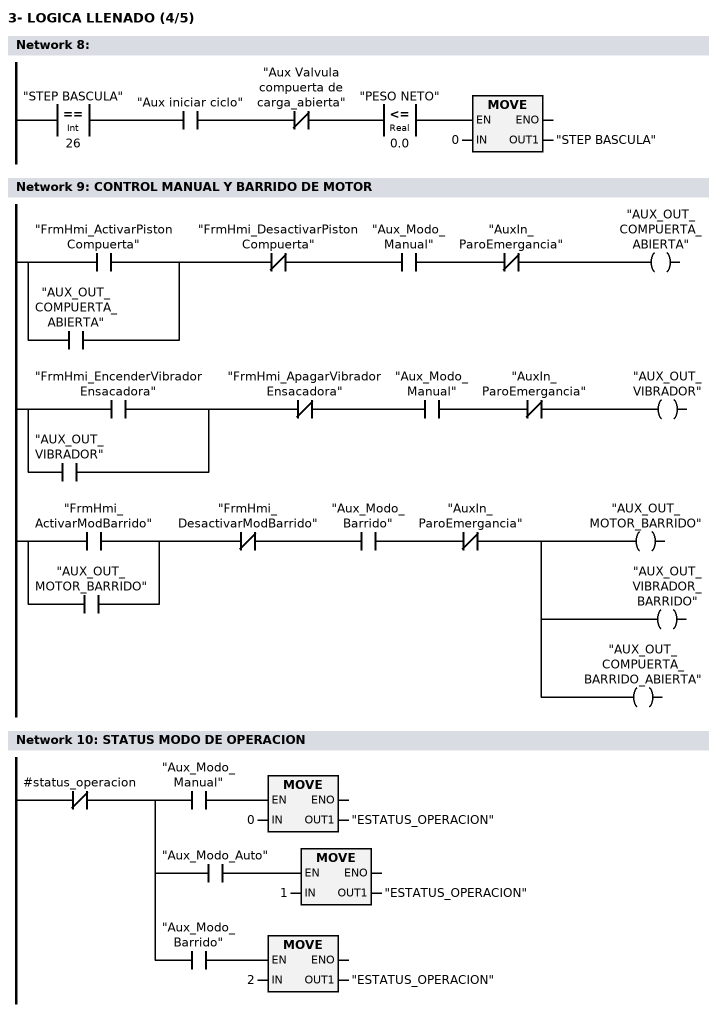
   RUNG wire#powerrail
      { S7_Templates := "SrcType := Int" } EQ_Contact(in1 := "STEP BASCULA", in2 := 26)
      Contact( "Aux iniciar ciclo" )
      I_Contact( "Aux Valvula compuerta de carga_abierta" )
      { S7_Templates := "SrcType := Real" } LE_Contact(in1 := "PESO NETO", in2 := 0.0)
      Move(in := 0, out1 => "STEP BASCULA")
   END_RUNG
   // the same network as SCL:
   IF ("STEP BASCULA" = 26) AND "Aux iniciar ciclo" AND NOT "Aux Valvula compuerta de carga_abierta" AND ("PESO NETO" <= 0.0) THEN
       "STEP BASCULA" := 0;
   END_IF;
END_REGION

REGION Network 9: CONTROL MANUAL Y BARRIDO DE MOTOR
   RUNG wire#powerrail
      Contact( "FrmHmi_ActivarPistonCompuerta" )
      wire#w1
      I_Contact( "FrmHmi_DesactivarPistonCompuerta" )
      Contact( "Aux_Modo_Manual" )
      I_Contact( "AuxIn_ParoEmergancia" )
      Coil( "AUX_OUT_COMPUERTA_ABIERTA" )
   END_RUNG
   RUNG wire#powerrail
      Contact( "AUX_OUT_COMPUERTA_ABIERTA" )
   END_RUNG wire#w1
   RUNG wire#powerrail
      Contact( "FrmHmi_EncenderVibradorEnsacadora" )
      wire#w2
      I_Contact( "FrmHmi_ApagarVibradorEnsacadora" )
      Contact( "Aux_Modo_Manual" )
      I_Contact( "AuxIn_ParoEmergancia" )
      Coil( "AUX_OUT_VIBRADOR" )
   END_RUNG
   RUNG wire#powerrail
      Contact( "AUX_OUT_VIBRADOR" )
   END_RUNG wire#w2
   RUNG wire#powerrail
      Contact( "FrmHmi_ActivarModBarrido" )
      wire#w3
      I_Contact( "FrmHmi_DesactivarModBarrido" )
      Contact( "Aux_Modo_Barrido" )
      I_Contact( "AuxIn_ParoEmergancia" )
      wire#w4
      Coil( "AUX_OUT_MOTOR_BARRIDO" )
   END_RUNG
   RUNG wire#powerrail
      Contact( "AUX_OUT_MOTOR_BARRIDO" )
   END_RUNG wire#w3
   RUNG wire#w4
      Coil( "AUX_OUT_VIBRADOR_BARRIDO" )
   END_RUNG
   RUNG wire#w4
      Coil( "AUX_OUT_COMPUERTA_BARRIDO_ABIERTA" )
   END_RUNG
   // the same network as SCL:
   "AUX_OUT_COMPUERTA_ABIERTA" := ("FrmHmi_ActivarPistonCompuerta" OR "AUX_OUT_COMPUERTA_ABIERTA") AND NOT "FrmHmi_DesactivarPistonCompuerta" AND "Aux_Modo_Manual" AND NOT "AuxIn_ParoEmergancia";
   "AUX_OUT_VIBRADOR" := ("FrmHmi_EncenderVibradorEnsacadora" OR "AUX_OUT_VIBRADOR") AND NOT "FrmHmi_ApagarVibradorEnsacadora" AND "Aux_Modo_Manual" AND NOT "AuxIn_ParoEmergancia";
   "AUX_OUT_MOTOR_BARRIDO" := ("FrmHmi_ActivarModBarrido" OR "AUX_OUT_MOTOR_BARRIDO") AND NOT "FrmHmi_DesactivarModBarrido" AND "Aux_Modo_Barrido" AND NOT "AuxIn_ParoEmergancia";
   "AUX_OUT_VIBRADOR_BARRIDO" := "AUX_OUT_MOTOR_BARRIDO";
   "AUX_OUT_COMPUERTA_BARRIDO_ABIERTA" := "AUX_OUT_MOTOR_BARRIDO";
END_REGION

REGION Network 10: STATUS MODO DE OPERACION
   RUNG wire#powerrail
      I_Contact( #status_operacion )
      wire#w1
      Contact( "Aux_Modo_Manual" )
      Move(in := 0, out1 => "ESTATUS_OPERACION")
   END_RUNG
   RUNG wire#w1
      Contact( "Aux_Modo_Auto" )
      Move(in := 1, out1 => "ESTATUS_OPERACION")
   END_RUNG
   RUNG wire#w1
      Contact( "Aux_Modo_Barrido" )
      Move(in := 2, out1 => "ESTATUS_OPERACION")
   END_RUNG
   // the same network as SCL:
   IF NOT #status_operacion AND "Aux_Modo_Manual" THEN "ESTATUS_OPERACION" := 0; END_IF;
   IF NOT #status_operacion AND "Aux_Modo_Auto" THEN "ESTATUS_OPERACION" := 1; END_IF;
   IF NOT #status_operacion AND "Aux_Modo_Barrido" THEN "ESTATUS_OPERACION" := 2; END_IF;
END_REGION

REGION Network 11: FALLAS
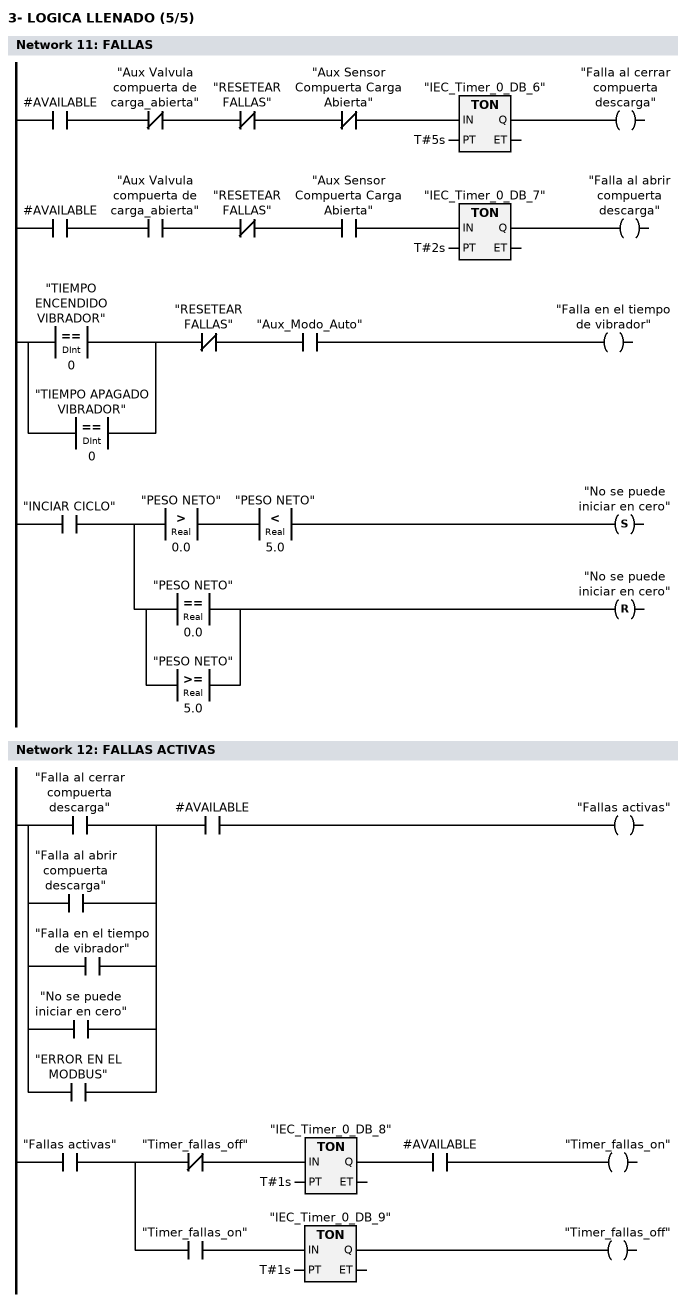
   "IEC_Timer_0_DB_6".TON(IN := #AVAILABLE AND NOT "Aux Valvula compuerta de carga_abierta" AND NOT "RESETEAR FALLAS" AND NOT "Aux Sensor Compuerta Carga Abierta",
                          PT := T#5s);
   "Falla al cerrar compuerta descarga" := "IEC_Timer_0_DB_6".Q;
   "IEC_Timer_0_DB_7".TON(IN := #AVAILABLE AND "Aux Valvula compuerta de carga_abierta" AND NOT "RESETEAR FALLAS" AND "Aux Sensor Compuerta Carga Abierta",
                          PT := T#2s);
   "Falla al abrir compuerta descarga" := "IEC_Timer_0_DB_7".Q;
   "Falla en el tiempo de vibrador" := (("TIEMPO ENCENDIDO VIBRADOR" = 0) OR ("TIEMPO APAGADO VIBRADOR" = 0)) AND NOT "RESETEAR FALLAS" AND "Aux_Modo_Auto";
   IF "INCIAR CICLO" AND ("PESO NETO" > 0.0) AND ("PESO NETO" < 5.0) THEN
       "No se puede iniciar en cero" := TRUE;
   END_IF;
   IF "INCIAR CICLO" AND (("PESO NETO" = 0.0) OR ("PESO NETO" >= 5.0)) THEN
       "No se puede iniciar en cero" := FALSE;
   END_IF;
END_REGION

REGION Network 12: FALLAS ACTIVAS
   "Fallas activas" := ("Falla al cerrar compuerta descarga" OR "Falla al abrir compuerta descarga" OR "Falla en el tiempo de vibrador" OR "No se puede iniciar en cero" OR "ERROR EN EL MODBUS") AND #AVAILABLE;
   "IEC_Timer_0_DB_8".TON(IN := "Fallas activas" AND NOT "Timer_fallas_off", PT := T#1s);
   "Timer_fallas_on" := "IEC_Timer_0_DB_8".Q AND #AVAILABLE;
   "IEC_Timer_0_DB_9".TON(IN := "Fallas activas" AND "Timer_fallas_on", PT := T#1s);
   "Timer_fallas_off" := "IEC_Timer_0_DB_9".Q;
END_REGION
END_ORGANIZATION_BLOCK

ORGANIZATION_BLOCK "4- SALIDAS"   // OB125, LAD, ProgramCycle
TITLE = "Main Program Sweep (Cycle)"
{ S7_Optimized_Access := 'TRUE' }
VERSION : 0.1
   VAR_INPUT
      Initial_Call : Bool;   // Initial call of this OB
      Remanence : Bool;   // =True, if remanent data are available
   END_VAR
   VAR_TEMP
      INHABILITADO : Bool;
      OUT : Bool;
   END_VAR
BEGIN

REGION Network 1: OUT VIBRADOR Y COMPUERTA
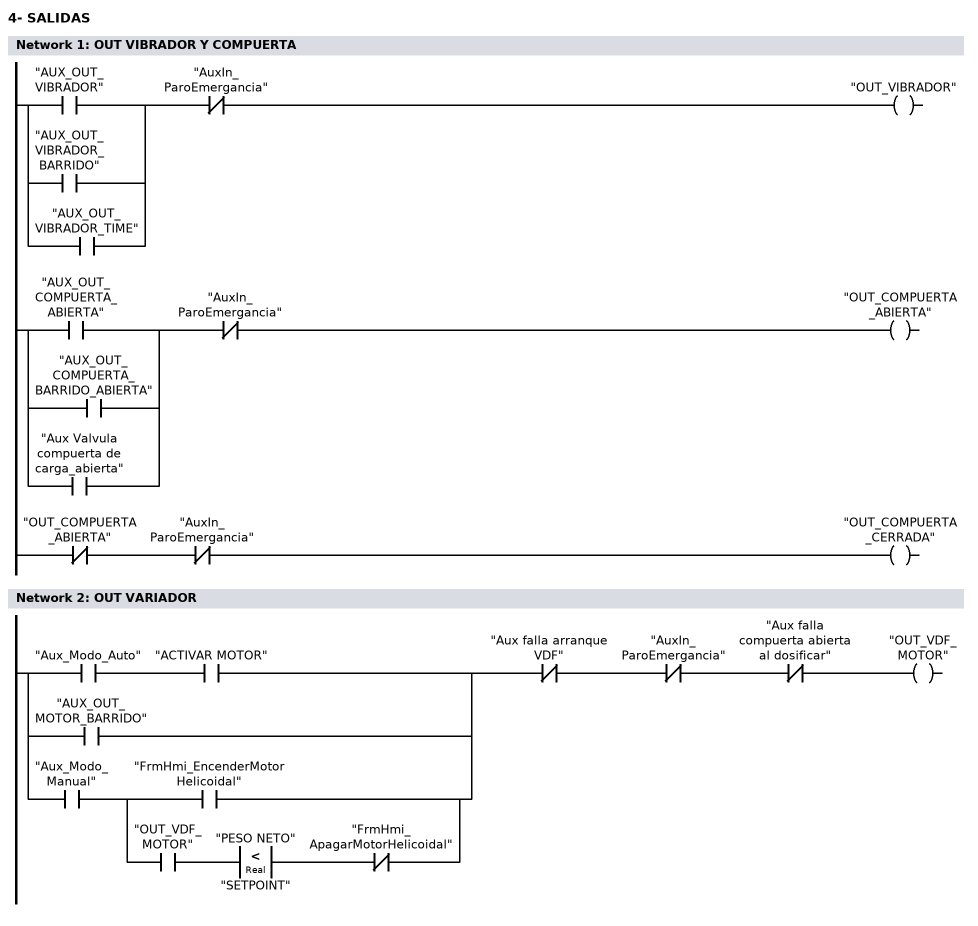
   RUNG wire#powerrail
      Contact( "AUX_OUT_VIBRADOR" )
      wire#w1
      I_Contact( "AuxIn_ParoEmergancia" )
      Coil( "OUT_VIBRADOR" )
   END_RUNG
   RUNG wire#powerrail
      Contact( "AUX_OUT_VIBRADOR_BARRIDO" )
   END_RUNG wire#w1
   RUNG wire#powerrail
      Contact( "AUX_OUT_VIBRADOR_TIME" )
   END_RUNG wire#w1
   RUNG wire#powerrail
      Contact( "AUX_OUT_COMPUERTA_ABIERTA" )
      wire#w2
      I_Contact( "AuxIn_ParoEmergancia" )
      Coil( "OUT_COMPUERTA_ABIERTA" )
   END_RUNG
   RUNG wire#powerrail
      Contact( "AUX_OUT_COMPUERTA_BARRIDO_ABIERTA" )
   END_RUNG wire#w2
   RUNG wire#powerrail
      Contact( "Aux Valvula compuerta de carga_abierta" )
   END_RUNG wire#w2
   RUNG wire#powerrail
      I_Contact( "OUT_COMPUERTA_ABIERTA" )
      I_Contact( "AuxIn_ParoEmergancia" )
      Coil( "OUT_COMPUERTA_CERRADA" )
   END_RUNG
   // the same network as SCL:
   "OUT_VIBRADOR" := ("AUX_OUT_VIBRADOR" OR "AUX_OUT_VIBRADOR_BARRIDO" OR "AUX_OUT_VIBRADOR_TIME") AND NOT "AuxIn_ParoEmergancia";
   "OUT_COMPUERTA_ABIERTA" := ("AUX_OUT_COMPUERTA_ABIERTA" OR "AUX_OUT_COMPUERTA_BARRIDO_ABIERTA" OR "Aux Valvula compuerta de carga_abierta") AND NOT "AuxIn_ParoEmergancia";
   "OUT_COMPUERTA_CERRADA" := NOT "OUT_COMPUERTA_ABIERTA" AND NOT "AuxIn_ParoEmergancia";
END_REGION

REGION Network 2: OUT VARIADOR
   RUNG wire#powerrail
      Contact( "Aux_Modo_Auto" )
      Contact( "ACTIVAR MOTOR" )
      wire#w1
      I_Contact( "Aux falla arranque VDF" )
      I_Contact( "AuxIn_ParoEmergancia" )
      I_Contact( "Aux falla compuerta abierta al dosificar" )
      Coil( "OUT_VDF_MOTOR" )
   END_RUNG
   RUNG wire#powerrail
      Contact( "AUX_OUT_MOTOR_BARRIDO" )
   END_RUNG wire#w1
   RUNG wire#powerrail
      Contact( "Aux_Modo_Manual" )
      wire#w2
      Contact( "FrmHmi_EncenderMotorHelicoidal" )
   END_RUNG wire#w1
   RUNG wire#w2
      Contact( "OUT_VDF_MOTOR" )
      { S7_Templates := "SrcType := Real" } LT_Contact(in1 := "PESO NETO", in2 := "SETPOINT")
      I_Contact( "FrmHmi_ApagarMotorHelicoidal" )
   END_RUNG wire#w1
   // the same network as SCL:
   "OUT_VDF_MOTOR" := (("Aux_Modo_Auto" AND "ACTIVAR MOTOR") OR "AUX_OUT_MOTOR_BARRIDO" OR ("Aux_Modo_Manual" AND ("FrmHmi_EncenderMotorHelicoidal" OR ("OUT_VDF_MOTOR" AND ("PESO NETO" < "SETPOINT") AND NOT "FrmHmi_ApagarMotorHelicoidal")))) AND NOT "Aux falla arranque VDF" AND NOT "AuxIn_ParoEmergancia" AND NOT "Aux falla compuerta abierta al dosificar";
END_REGION
END_ORGANIZATION_BLOCK

ORGANIZATION_BLOCK "5- CALIBRACION"   // OB126, LAD, ProgramCycle
TITLE = "Main Program Sweep (Cycle)"
{ S7_Optimized_Access := 'TRUE' }
VERSION : 0.1
   VAR_INPUT
      Initial_Call : Bool;   // Initial call of this OB
      Remanence : Bool;   // =True, if remanent data are available
   END_VAR
BEGIN

REGION Network 1: VER CALIBRACION EN HMI
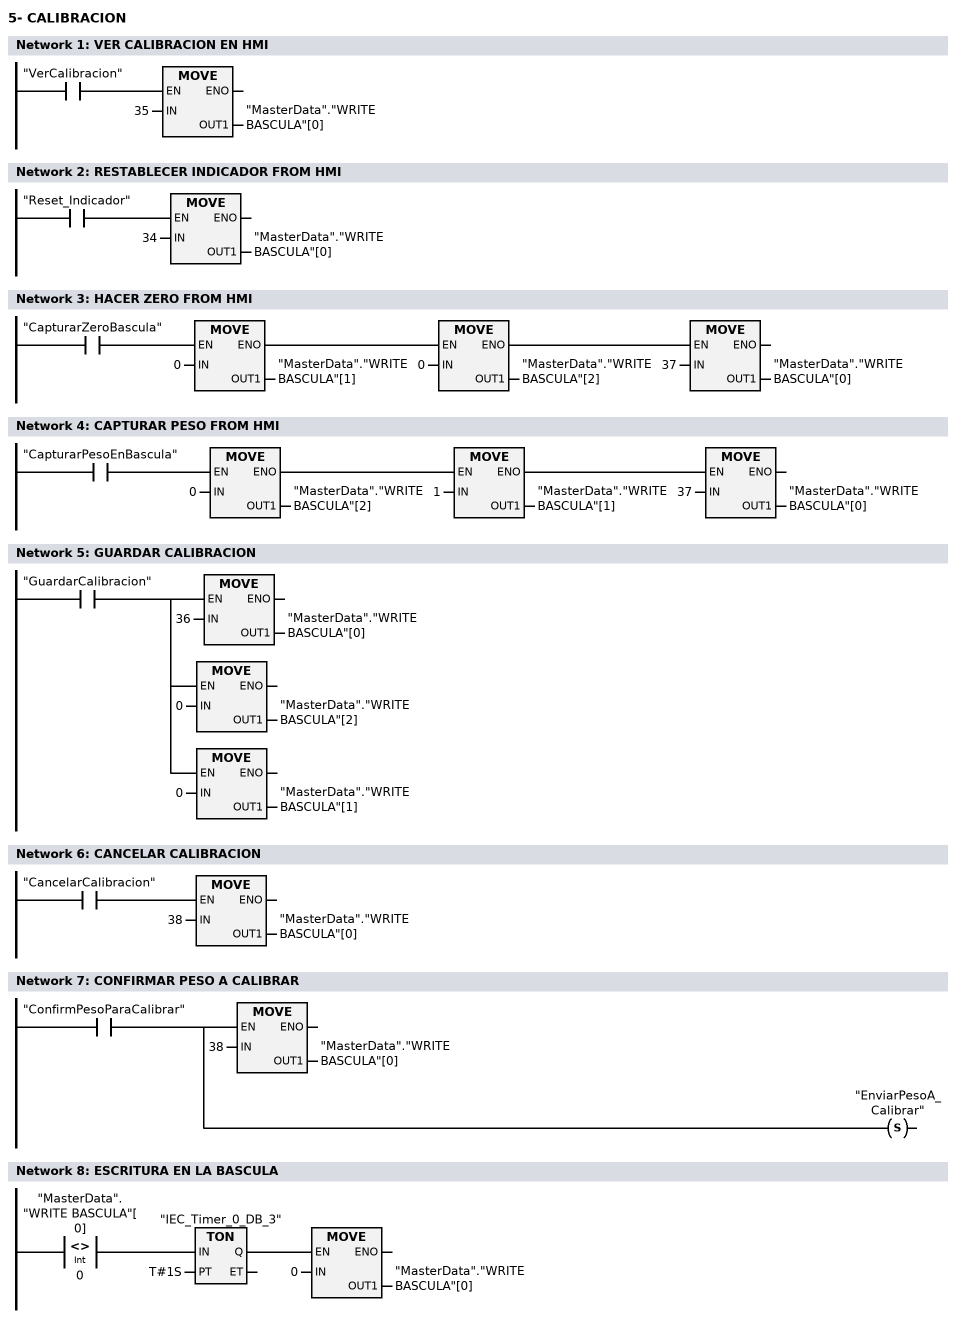
   RUNG wire#powerrail
      Contact( "VerCalibracion" )
      Move(in := 35, out1 => "MasterData"."WRITE BASCULA"[0])
   END_RUNG
   // the same network as SCL:
   IF "VerCalibracion" THEN "MasterData"."WRITE BASCULA"[0] := 35; END_IF;
END_REGION

REGION Network 2: RESTABLECER INDICADOR FROM HMI
   RUNG wire#powerrail
      Contact( "Reset_Indicador" )
      Move(in := 34, out1 => "MasterData"."WRITE BASCULA"[0])
   END_RUNG
   // the same network as SCL:
   IF "Reset_Indicador" THEN "MasterData"."WRITE BASCULA"[0] := 34; END_IF;
END_REGION

REGION Network 3: HACER ZERO FROM HMI
   RUNG wire#powerrail
      Contact( "CapturarZeroBascula" )
      Move(in := 0, out1 => "MasterData"."WRITE BASCULA"[1])
      Move(in := 0, out1 => "MasterData"."WRITE BASCULA"[2])
      Move(in := 37, out1 => "MasterData"."WRITE BASCULA"[0])
   END_RUNG
   // the same network as SCL:
   IF "CapturarZeroBascula" THEN
       "MasterData"."WRITE BASCULA"[1] := 0;
       "MasterData"."WRITE BASCULA"[2] := 0;
       "MasterData"."WRITE BASCULA"[0] := 37;
   END_IF;
END_REGION

REGION Network 4: CAPTURAR PESO FROM HMI
   RUNG wire#powerrail
      Contact( "CapturarPesoEnBascula" )
      Move(in := 0, out1 => "MasterData"."WRITE BASCULA"[2])
      Move(in := 1, out1 => "MasterData"."WRITE BASCULA"[1])
      Move(in := 37, out1 => "MasterData"."WRITE BASCULA"[0])
   END_RUNG
   // the same network as SCL:
   IF "CapturarPesoEnBascula" THEN
       "MasterData"."WRITE BASCULA"[2] := 0;
       "MasterData"."WRITE BASCULA"[1] := 1;
       "MasterData"."WRITE BASCULA"[0] := 37;
   END_IF;
END_REGION

REGION Network 5: GUARDAR CALIBRACION
   RUNG wire#powerrail
      Contact( "GuardarCalibracion" )
      wire#w1
      Move(in := 36, out1 => "MasterData"."WRITE BASCULA"[0])
   END_RUNG
   RUNG wire#w1
      Move(in := 0, out1 => "MasterData"."WRITE BASCULA"[2])
   END_RUNG
   RUNG wire#w1
      Move(in := 0, out1 => "MasterData"."WRITE BASCULA"[1])
   END_RUNG
   // the same network as SCL:
   IF "GuardarCalibracion" THEN
       "MasterData"."WRITE BASCULA"[0] := 36;
       "MasterData"."WRITE BASCULA"[2] := 0;
       "MasterData"."WRITE BASCULA"[1] := 0;
   END_IF;
END_REGION

REGION Network 6: CANCELAR CALIBRACION
   RUNG wire#powerrail
      Contact( "CancelarCalibracion" )
      Move(in := 38, out1 => "MasterData"."WRITE BASCULA"[0])
   END_RUNG
   // the same network as SCL:
   IF "CancelarCalibracion" THEN "MasterData"."WRITE BASCULA"[0] := 38; END_IF;
END_REGION

REGION Network 7: CONFIRMAR PESO A CALIBRAR
   RUNG wire#powerrail
      Contact( "ConfirmPesoParaCalibrar" )
      wire#w1
      Move(in := 38, out1 => "MasterData"."WRITE BASCULA"[0])
   END_RUNG
   RUNG wire#w1
      S_Coil( "EnviarPesoA_Calibrar" )
   END_RUNG
   // the same network as SCL:
   IF "ConfirmPesoParaCalibrar" THEN
       "MasterData"."WRITE BASCULA"[0] := 38;
       "EnviarPesoA_Calibrar" := TRUE;
   END_IF;
END_REGION

REGION Network 8: ESCRITURA EN LA BASCULA
   "IEC_Timer_0_DB_3".TON(IN := "MasterData"."WRITE BASCULA"[0] <> 0, PT := T#1S);
   IF "IEC_Timer_0_DB_3".Q THEN "MasterData"."WRITE BASCULA"[0] := 0; END_IF;
END_REGION
END_ORGANIZATION_BLOCK

ORGANIZATION_BLOCK "6- CONTADOR"   // OB127, LAD, ProgramCycle
TITLE = "Main Program Sweep (Cycle)"
{ S7_Optimized_Access := 'TRUE' }
VERSION : 0.1
   VAR_INPUT
      Initial_Call : Bool;   // Initial call of this OB
      Remanence : Bool;   // =True, if remanent data are available
   END_VAR
   VAR_TEMP
      available : Bool;
      "TIME ON" : Time;
      "TIME OFF" : Time;
      "RESULTADO MUL OFF" : Int;
      "RESULTADO MUL ON" : Int;
   END_VAR
BEGIN

REGION Network 1: CONTADOR DE PRUEBA
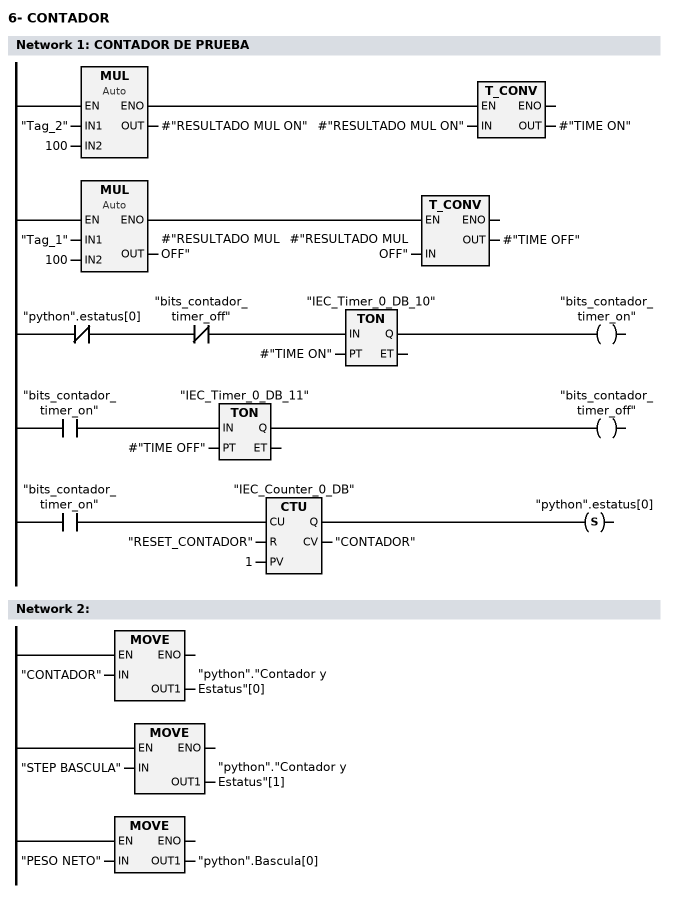
   #"RESULTADO MUL ON" := "Tag_2" * 100;
   #"TIME ON" := T_CONV(IN := #"RESULTADO MUL ON");
   #"RESULTADO MUL OFF" := "Tag_1" * 100;
   #"TIME OFF" := T_CONV(IN := #"RESULTADO MUL OFF");
   "IEC_Timer_0_DB_10".TON(IN := NOT "python".estatus[0] AND NOT "bits_contador_timer_off", PT := #"TIME ON");
   "bits_contador_timer_on" := "IEC_Timer_0_DB_10".Q;
   "IEC_Timer_0_DB_11".TON(IN := "bits_contador_timer_on", PT := #"TIME OFF");
   "bits_contador_timer_off" := "IEC_Timer_0_DB_11".Q;
   "IEC_Counter_0_DB".CTU(CU := "bits_contador_timer_on", R := "RESET_CONTADOR", PV := 1, CV => "CONTADOR");
   IF "IEC_Counter_0_DB".Q THEN "python".estatus[0] := TRUE; END_IF;
END_REGION

REGION Network 2
   RUNG wire#powerrail
      Move(in := "CONTADOR", out1 => "python"."Contador y Estatus"[0])
   END_RUNG
   RUNG wire#powerrail
      Move(in := "STEP BASCULA", out1 => "python"."Contador y Estatus"[1])
   END_RUNG
   RUNG wire#powerrail
      Move(in := "PESO NETO", out1 => "python".Bascula[0])
   END_RUNG
   // the same network as SCL:
   "python"."Contador y Estatus"[0] := "CONTADOR";
   "python"."Contador y Estatus"[1] := "STEP BASCULA";
   "python".Bascula[0] := "PESO NETO";
END_REGION
END_ORGANIZATION_BLOCK